METHOD ErrorHandler : BOOL
VAR_INPUT
END_VAR
VAR
END_VAR
//once error scanned
IF currentMode = eOperationModes.AUTO THEN
	//once error deteted and in AUTO mode , forcely switch to SEMI_AUTO
	currentMode := eOperationModes.SEMI_AUTO;
END_IF
//reset error handling
IF requestErrorClear <> eErrorClearWays.NO_ACTION THEN
	errorDevice^.ErrorClear(requestErrorClear); //call error clear function
	requestErrorClear := eErrorClearWays.NO_ACTION;
	errorDevice := 0 ;// cut link
END_IF
END_METHOD

METHOD FB_init : BOOL
VAR_INPUT
	bInitRetains : BOOL; // if TRUE, the retain variables are initialized (warm start / cold start)
	bInCopyCode : BOOL;  // if TRUE, the instance afterwards gets moved into the copy code (online change)
	
	argParent : POINTER TO RunUnitGeneric;
	argSlotBase : POINTER TO RunMaterial;
	argSlotLast : POINTER TO RunMaterial;
	
	argPbRed : POINTER TO RunSignal;
	argPbGreen : POINTER TO RunSignal;
	argPbYellow : POINTER TO RunSignal;
	
	argInterfaceControl : POINTER TO InterfaceControlV1;
	argInterfaceManual : POINTER TO InterfaceManualV1;
END_VAR
//initialize 
Parent := argParent;
SlotBase := argSlotBase;
SlotLast := argSlotLast;
//
IF bInitRetains THEN
	NextState := eSpecialStates.INITIAL_BEGIN;
END_IF
//input
pbRed := argPbRed;
pbGreen := argPbGreen;
pbYellow := argPbYellow;

interfaceControl := argInterfaceControl;
interfaceManual := argInterfaceManual;

interfaceControl^.state := TO_WORD(eSpecialStates.MAIN_WAIT_INITIALIZING);
END_METHOD

METHOD Initialize : BOOL
VAR_INPUT
END_VAR
END_METHOD

END_FUNCTION_BLOCK

// ---- POUs/Foundation/RunUnitIndexerMaster.TcPOU
FUNCTION_BLOCK RunUnitIndexerMaster EXTENDS RunUnitTransporterBase
VAR		
	Axis : POINTER TO RunAxis; //axis reference
	
	//Working registers
	nCounter : DINT;
	
	
END_VAR
VAR PERSISTENT
END_VAR

SUPER^(); // call base class's execution

//---------------
//	S16#0-S16#0F : regular state as standard indexer
//	S16#10 : mechanical control of movement
//---------------

IF NOT workingTimer.IN THEN
	 workingTimer.IN := TRUE;
END_IF

CASE outputState OF
	16#0:
		//-------------------------
		//	Trigger all slaves
		//-------------------------
		FOR nCounter:=1 TO 4 BY 1 DO
			slaveWorkingSignal[nCounter] := slaveLinkageStatus[nCounter];
		END_FOR
		bSerialTransition := TRUE;
		
		THIS^.workingTimerCache := THIS^.workingTimer.ET;
		workingTimer.IN := FALSE; //reset
	16#1:	
		//------------------------------------------
		//check material synchronization to Databse
		//All slot act must be off
		//------------------------------------------
		bSerialTransition := TRUE;
		FOR nCounter:=0 TO SlotCount-1 BY 1 DO
			bSerialTransition := bSerialTransition AND NOT SlotBase[nCounter].Act;
		END_FOR
	16#2:
		//--------------------------------
		// Scanning working signal until all are off
		//--------------------------------
		bSerialTransition := TRUE;
		FOR nCounter:= 1 TO 32 BY 1 DO
			bSerialTransition := bSerialTransition AND NOT slaveWorkingSignal[nCounter];
		END_FOR
	16#3:
		//-------------------
		//Sync with down stream
		//-------------------
		IF syncEngaged AND syncAcknowledged THEN
			syncEngaged := FALSE; //reset
		END_IF
		bSerialTransition := NOT syncAcknowledged; //make sure signal is resetted
		IF bSerialTransition THEN
			//move last slot's information to buffer area
			syncMatId:= SlotLast^.Id; // for the last slot
			syncMatValid := SlotLast^.Valid;// ready to sync
		END_IF
	16#4:
		//2 modes
		// a. synchronize with downstream only, go with pull upstream if avialable
		// b. synchronize with down/upstream both
	
		// pull by downstream (set on then check off
		// pull upstream (check on then reset
		
		IF syncMatValid AND NOT syncEngaged THEN
			syncEngaged := TRUE;//ready to synchronizing (communicate with downstream
		END_IF
		
		//listen to move
		bSerialTransition :=  (NOT syncMatValid) OR (syncAcknowledged AND syncMatValid);
		IF bSerialTransition THEN
			NextState := 16#10;
		END_IF
	16#10:
		//---------------------
		//shifting movement mechaincal
		//---------------------	
	16#F:
		//---------------------------------------------------------------
		//Do data shifting (move is valid/id) , leave first slot as empty
		//---------------------------------------------------------------
		FOR nCounter:=SlotCount-1 TO 0 BY -1 DO
			IF nCounter > 0 THEN
				SlotBase[nCounter].Id := SlotBase[nCounter-1].id;
				SlotBase[nCounter].Valid := SlotBase[nCounter-1].Valid;
			END_IF			
		END_FOR
		NextState := 16#0;
END_CASE

METHOD FB_init : BOOL
VAR_INPUT
	bInitRetains : BOOL; // if TRUE, the retain variables are initialized (warm start / cold start)
	bInCopyCode : BOOL;  // if TRUE, the instance afterwards gets moved into the copy code (online change)
	
	argParent : POINTER TO RunUnitGeneric;
	argSlotBase : POINTER TO RunMaterial;
	argSlotLast : POINTER TO RunMaterial;
	
	argUpstream : POINTER TO RunUnitTransporterBase;
	argAxis : POINTER TO RunAxis;

END_VAR
//initialize 
Parent := argParent;
SlotBase := argSlotBase;
SlotLast := argSlotLast;

Axis := argAxis;
Upstream := argUpstream;

IF Upstream=0 THEN
	isProxyMode:=TRUE; //no upstream , i am proxy
END_IF

//calculate how much slot related
SlotCount :=  TO_INT((SlotLast-SlotBase)/SIZEOF(RunMaterial) + 1);
END_METHOD

END_FUNCTION_BLOCK

// ---- POUs/Foundation/RunUnitTransporterBase.TcPOU
FUNCTION_BLOCK RunUnitTransporterBase EXTENDS RunUnitGeneric
VAR_INPUT	
	//self
	syncAcknowledged AT%M*  : BOOL; //downstream replied starting ackowledge , face to downstream
	syncMatId AT%M* : DWORD := 0;
	syncMatValid AT%M* : BOOL := FALSE;
END_VAR
VAR_OUTPUT
	//self
	syncEngaged AT%M*  : BOOL; //inform downstream i am ready , face to downstream
	
END_VAR
VAR		
	//
	Upstream : POINTER TO RunUnitTransporterBase;//upstream linkage
	//proxy mode
	isProxyMode : BOOL := FALSE;
	
	pollingTimer : TON;
	fbAdsSyncRead : FB_ReadAdsSymByName;
	fbAdsSyncWrite : FB_WriteAdsSymByName;
	fbAdsSyncMatIdRead : FB_ReadAdsSymByName;
	fbAdsSyncMatValidRead : FB_ReadAdsSymByName;
	
	preSyncEngaged : BOOL := FALSE;
	
END_VAR
VAR PERSISTENT
	//proxy mode parameters
	netId : T_AmsNetID;
	port : T_AmsPort := 851; //Tc3
	
	varNameSyncEngaged : STRING;
	varNameSyncAckowledged : STRING;
	varNameSyncMatIdSync : STRING;
	varNameSyncMatValidSync : STRING;
END_VAR

//non proxy 	
SUPER^();

IF (outputState <> NextState) OR bSerialTransition THEN
	//once state transit , reset timer
	timeoutTimer.IN := FALSE;
ELSIF NOT timeoutTimer.IN THEN
	//once timer not activated 
	timeoutTimer.IN := TRUE;
END_IF

IF NOT isProxyMode THEN
	RETURN;
END_IF

pollingTimer(IN:= NOT pollingTimer.Q, PT:= T#50MS, Q=> , ET=> );

//do ADS data exchanging
fbAdsSyncRead(
	bRead:= pollingTimer.Q and not fbAdsSyncRead.bBusy, 
	sNetId:= netId, 
	nPort:= port, 
	sVarName:= varNameSyncEngaged, 
	nDestAddr:= ADR(preSyncEngaged), 
	nLen:= SIZEOF(preSyncEngaged), 
	tTimeout:= , 
	eComMode:= , 
	bBusy=> , 
	bError=> , 
	nErrorId=> );
		
fbAdsSyncWrite(
	bWrite:= pollingTimer.Q AND NOT fbAdsSyncWrite.bBusy, 
	sNetId:= netId, 
	nPort:= port, 
	sVarName:= varNameSyncAckowledged, 
	nSrcAddr:= ADR(syncAcknowledged), 
	nLen:= SIZEOF(syncAcknowledged), 
	tTimeout:= , 
	eComMode:= , 
	bBusy=> , 
	bError=> , 
	nErrorId=> );		
			
fbAdsSyncMatIdRead(
	bRead:= , 
	sNetId:= netId, 
	nPort:= port, 
	sVarName:= varNameSyncMatIdSync, 
	nDestAddr:= ADR(syncMatId), 
	nLen:= SIZEOF(syncMatId), 
	tTimeout:= , 
	eComMode:= , 
	bBusy=> , 
	bError=> , 
	nErrorId=> );
fbAdsSyncMatValidRead(
	bRead:= , 
	sNetId:= netId, 
	nPort:= port, 
	sVarName:= varNameSyncMatValidSync, 
	nDestAddr:= ADR(syncMatValid), 
	nLen:= SIZEOF(syncMatValid), 
	tTimeout:= , 
	eComMode:= , 
	bBusy=> , 
	bError=> , 
	nErrorId=> );
	

//data exchanging do not be break
atomicOperation := TRUE;
CASE outputState OF
	0:
		IF preSyncEngaged THEN
						
			//start reading
			fbAdsSyncMatIdRead.bRead := TRUE;
			fbAdsSyncMatValidRead.bRead:= TRUE;
			
			bSerialTransition := TRUE;
		END_IF
	1:
		IF NOT fbAdsSyncMatIdRead.bBusy AND NOT fbAdsSyncMatValidRead.bBusy THEN
			syncEngaged:= TRUE; //mat sync verified , output to downstream
			bSerialTransition := TRUE;
		END_IF
	2: 
		IF NOT preSyncEngaged THEN
			//done
			syncEngaged := FALSE;
			//wait for next reading
			fbAdsSyncMatIdRead.bRead := FALSE;
			fbAdsSyncMatValidRead.bRead:= FALSE;
			
			
			NextState := 0;
		END_IF
END_CASE

METHOD FB_init : BOOL
VAR_INPUT
	bInitRetains : BOOL; // if TRUE, the retain variables are initialized (warm start / cold start)
	bInCopyCode : BOOL;  // if TRUE, the instance afterwards gets moved into the copy code (online change)
	
	argParent : POINTER TO RunUnitGeneric;
	argSlotBase : POINTER TO RunMaterial;
	argSlotLast : POINTER TO RunMaterial;
	
	argUpstream : POINTER TO RunUnitTransporterBase;
END_VAR
//initialize 
Parent := argParent;
SlotBase := argSlotBase;
SlotLast := argSlotLast;

Upstream := argUpstream;

IF Upstream=0 THEN
	isProxyMode:=TRUE; //no upstream , i am proxy
END_IF
END_METHOD

METHOD Initialize : BOOL
VAR_INPUT
END_VAR

//reset sync signal
CASE outputState OF
	eSpecialStates.INITIAL_BEGIN:
		syncEngaged := FALSE; //reset
		IF Upstream <> 0 THEN
			Upstream^.syncAcknowledged := FALSE; //reset
		END_IF
		//direct change state
		NextState := eSpecialStates.INITIAL_END;
END_CASE

Initialize := SUPER^.Initialize();
END_METHOD

END_FUNCTION_BLOCK

// ---- POUs/IncNoOverflow.TcPOU
FUNCTION IncNoOverflow : UDINT
VAR_INPUT
	input : UDINT;
END_VAR
VAR
END_VAR

IF input >= 16#FFFFFFFF THEN
	IncNoOverflow := 0;
ELSE
	IncNoOverflow := input +1;
END_IF

END_FUNCTION

// ---- POUs/MAIN.TcPOU
PROGRAM MAIN
VAR

cbBlock1 : CommandBlockBase;
cbBlock2 : CommandBlockBase;

cbBlock3 : CommandBlockPos;
cbBlock4 : CommandBlockPos;

ptBlock : POINTER TO CommandBlockBase := ADR(cbBlock1);	
ptBlockPos : POINTER TO CommandBlockPos;

aSize : INT;


memoryPool : ARRAY[1..1024] OF WORD;

ptRunIndexerMaster : POINTER TO RunUnitIndexerMaster;
ptRunGeneric : POINTER TO RunUnitGeneric;

ptUnitGeneric : POINTER TO UnitBase;
ptUnitIndexerMaster : POINTER TO UnitIndexerMaster;

bInitialized : BOOL ;
nCounter : int ;
END_VAR

cbBlock1.AXIS_ID:=5;
MAIN.ptBlock:=ADR(cbBlock1);

cbBlock2:=MAIN.ptBlock^; // value assignment?
//change cbBlock1 , watch if cbBlock2 changed

MAIN.ptBlock := ADR(cbBlock3); //if possible mophism

cbBlock3.COORDINATE:=1234;

ptBlockPos:=MAIN.ptBlock;
cbBlock4:=ptBlockPos^;//check


//may access violation??
//ptBlockPos:=ADR(cbBlock1);
//ptBlockPos^.COORDINATE:=5555; //may violation

//TEST2();
//TEST_CYLINDER();
//TEST_UNIT_VIRTUAL();
//TEST_UNIT_MASTER();
//TEST_AXIS();
IF NOT bInitialized THEN
	FOR nCounter:=8 TO 10 BY 1 DO
		GVL.commandBlocks[nCounter].command := eCommandTypes.POSITION;
		GVL.commandBlocks[nCounter].parameter.position.Acceleration := 4000;
		GVL.commandBlocks[nCounter].parameter.position.Deceleration := 4000;

	END_FOR
	GVL.commandBlocks[8].parameter.position.Position := 300;
	GVL.commandBlocks[8].parameter.position.Velocity := 400;
	
	GVL.commandBlocks[9].parameter.position.Position := 400;
	GVL.commandBlocks[9].parameter.position.Velocity := 100;
	
	GVL.commandBlocks[10].parameter.position.Position := 800;
	GVL.commandBlocks[10].parameter.position.Velocity := 400;
	
	bInitialized := true;
END_IF
TEST_BUFFERING();

aSize := SIZEOF(GVL.unitControls[1]);
aSize := SIZEOF(UnitBase);
aSize := SIZEOF(UnitIndexerMaster);
//fbCylinder(ptBlock:= ADR(cylinderBlock));

//fbRunIndexerMaster(ptBlock:= );


//no need
//ptRunIndexerMaster := ADR(memoryPool[1]); // fine?
//ptRunGeneric := ADR(memoryPool[1+SIZEOF(ptRunIndexerMaster)]);

//ptRunIndexerMaster^();
//ptRunGeneric^();


//possible manipulate memory allocation
ptUnitGeneric := ADR(memoryPool[1]);
ptUnitIndexerMaster := ADR(memoryPool[1+SIZEOF(ptUnitGeneric^)]);

ptUnitGeneric^.alarmCode := 99;  //

METHOD FB_init : BOOL
VAR_INPUT
	bInitRetains : BOOL; // if TRUE, the retain variables are initialized (warm start / cold start)
	bInCopyCode : BOOL;  // if TRUE, the instance afterwards gets moved into the copy code (online change)
END_VAR
END_METHOD

END_PROGRAM

// ---- POUs/Stations/CellularD/RunCableHolder.TcPOU
FUNCTION_BLOCK RunCableHolder EXTENDS RunUnitSlave
VAR
	//devices
	holderFixedEnd : POINTER TO RunCylinder;
	holderMovingEnd : POINTER TO RunCylinder;
	shifterShort : POINTER TO RunCylinder;
	shifterLong : POINTER TO RunCylinder;
	//axis (share
	axis : POINTER TO RunAxis;
	ptDrag : POINTER TO ParameterSet;
	ptRelease : pointer to ParameterSet;
END_VAR

SUPER^();

CASE outputState OF
	//---------------Initialize
	eSpecialStates.INITIAL_BEGIN:
		transitionByte.0 :=  holderFixedEnd^.Execute(eCylinderCommands.COMMAND_A);
		transitionByte.1 :=  holderMovingEnd^.Execute(eCylinderCommands.COMMAND_A);
		transitionByte.2 :=  shifterShort^.Execute(eCylinderCommands.COMMAND_A);
		transitionByte.3 :=  shifterLong^.Execute(eCylinderCommands.COMMAND_A);
		IF transitionByte = 16#F THEN
			NextState := eSpecialStates.INITIAL_END;
		END_IF
	//---------------Working
	eSpecialStates.SLAVE_ENTER_PROCEDURE:
		IF bMaterialOverride THEN
			bSerialTransition := TRUE;
		ELSE
			NextState := eSpecialStates.SLAVE_WORK_DONE;	
		END_IF
		//TODO , check ok/ng?
	16#201:
		bSerialTransition := shifterLong^.Execute(eCylinderCommands.COMMAND_B);
	16#202:
		//hold
		transitionByte.0 :=  holderFixedEnd^.Execute(eCylinderCommands.COMMAND_B);
		transitionByte.1 :=  holderMovingEnd^.Execute(eCylinderCommands.COMMAND_B);
		bSerialTransition := (transitionByte = 16#3);
	16#203:
		bSerialTransition := axis^.ExecuteParameter(ptDrag);//inform transporter moving work2
	16#204:
		//strech
		IF shifterShort^.Execute(eCylinderCommands.COMMAND_B) THEN
			slaveWorkingSignal[1] := TRUE; //inform to labeler handler to work
			NextState := 16#210;
		END_IF
	//-------------Releasing
	16#210:
		//wait until
		bSerialTransition := NOT slaveWorkingSignal[1];
	16#211:
		transitionByte.0 := holderFixedEnd^.Execute(eCylinderCommands.COMMAND_A); //release
		transitionByte.1 := holderMovingEnd^.Execute(eCylinderCommands.COMMAND_A);
		IF transitionByte = 16#3 THEN
			bSerialTransition := TRUE;
		END_IF
	16#212:
		bSerialTransition := axis^.ExecuteParameter(ptRelease);//inform transporter moving release
	16#213:
		//release
		bSerialTransition := shifterLong^.Execute(eCylinderCommands.COMMAND_A);
	16#214:
		//release
		bSerialTransition := holderMovingEnd^.Execute(eCylinderCommands.COMMAND_A);
	16#215:
		IF shifterShort^.Execute(eCylinderCommands.COMMAND_A) THEN
			NextState := eSpecialStates.SLAVE_WORK_DONE; //rewind
		END_IF
END_CASE

METHOD FB_init : BOOL
VAR_INPUT
	bInitRetains : BOOL; // if TRUE, the retain variables are initialized (warm start / cold start)
	bInCopyCode : BOOL;  // if TRUE, the instance afterwards gets moved into the copy code (online change)
	
	argParent : POINTER TO RunUnitGeneric;
	argSlotBase : POINTER TO RunMaterial;
	argSlotLast : POINTER TO RunMaterial;
	
	argWorkingSignal : POINTER TO BOOL;
	
	//devices
	argHolderFixedEnd : POINTER TO RunCylinder;
	argHolderMovingEnd : POINTER TO RunCylinder;
	argShifterShort : POINTER TO RunCylinder;
	argShifterLong : POINTER TO RunCylinder;
	
	//
	argAxis : POINTER TO RunAxis;
END_VAR
VAR CONSTANT
	indexDrag : INT :=8;
	indexRelease : int :=9;
END_VAR
//initialize 
Parent := argParent;
SlotBase := argSlotBase;
SlotLast := argSlotLast;
//
IF bInitRetains THEN
	NextState := eSpecialStates.INITIAL_BEGIN;
END_IF

workingSignal := argWorkingSignal; //link

//device link
holderFixedEnd := argHolderFixedEnd;
holderMovingEnd := argHolderMovingEnd;
shifterShort := argShifterShort;
shifterLong := argShifterLong;

//
axis := argAxis;
ptDrag := ADR(axis^.ptpCommands[indexDrag]);
ptRelease := ADR(axis^.ptpCommands[indexRelease]);
END_METHOD

END_FUNCTION_BLOCK

// ---- POUs/Stations/CellularD/RunGradeOutput.TcPOU
FUNCTION_BLOCK RunGradeOutput EXTENDS RunUnitSlave
VAR
	axisMoving : POINTER TO RunAxis;
	holder : POINTER TO RunCylinder;
	axisVertical : POINTER TO RunCylinder;
	clamper : POINTER TO RunCylinder;	
	//
	ptCommandReady : POINTER TO ParameterSet;
	ptCommandOK : POINTER TO ParameterSet;
	ptCommandNG : POINTER TO ParameterSet;
	//
	block : MaterialBlock;
	ptDesitination : POINTER TO parameterset;
END_VAR
VAR PERSISTENT
	isQuery : bool ; //whether query material data when material income
END_VAR

//Ng/OK output mechanism
SUPER^();

CASE outputState OF 
	//-------------------------Initialize
	eSpecialStates.INITIAL_BEGIN:
		transitionByte.0 := holder^.Execute(eCylinderCommands.COMMAND_A);
		transitionByte.1 := clamper^.Execute(eCylinderCommands.COMMAND_A);
		bSerialTransition := (transitionByte = 16#3);
	eSpecialStates.INITIAL_STATE_1:
		bSerialTransition :=  axisVertical^.Execute(eCylinderCommands.COMMAND_A);
	eSpecialStates.INITIAL_STATE_2:
		IF axisMoving^.ExecuteParameter(ptCommandReady) THEN
			NextState := eSpecialStates.INITIAL_END;
		END_IF
	//------------------------Working
	eSpecialStates.SLAVE_ENTER_PROCEDURE:
		//---------------
		//	Material infor exchanging
		//---------------
		SlotLast^.Id := SlotBase^.Id; //the clamper work station
		SlotLast^.Valid := SlotLast^.Valid;
		IF SlotLast^.Valid THEN
			SlotLast^.Act := isQuery; //query grade
			bSerialTransition := TRUE;
		ELSE
			NextState := eSpecialStates.SLAVE_WORK_DONE;		
		END_IF
	16#201:
		bSerialTransition:=axisVertical^.Execute(eCylinderCommands.COMMAND_B); //down
	16#202:
		bSerialTransition:=holder^.Execute(eCylinderCommands.COMMAND_B); //hold
	16#203:
		bSerialTransition:=clamper^.Execute(eCylinderCommands.COMMAND_B); //clamper relase
	16#204:
		bSerialTransition:=axisVertical^.Execute(eCylinderCommands.COMMAND_A); //up
	16#205:
		bSerialTransition:=clamper^.Execute(eCylinderCommands.COMMAND_A); //clamper return
		IF bSerialTransition THEN
			workingSignal^ := FALSE; //release conveyor
		END_IF
	16#206:
		bSerialTransition := NOT SlotLast^.Act; //wait until query over
		IF bSerialTransition THEN
			block := SlotLast^.Data;
			CASE block.data[0] OF
				0:
					//ng
					ptDesitination := ptCommandNG;
				1:
					//ok
					ptDesitination := ptCommandOK;
			END_CASE
		END_IF
	16#207:
		IF axisMoving^.ExecuteParameter(ptDesitination) THEN
			//according TO grade TO MOVE
			NextState := 16#210;
		END_IF
	//-------------------Drop
	16#210: 
		bSerialTransition:=holder^.Execute(eCylinderCommands.COMMAND_A); //release
	16#211:
		IF axisMoving^.ExecuteParameter(ptCommandReady) THEN
			NextState := 0;
		END_IF
END_CASE

METHOD FB_init : BOOL
VAR_INPUT
	bInitRetains : BOOL; // if TRUE, the retain variables are initialized (warm start / cold start)
	bInCopyCode : BOOL;  // if TRUE, the instance afterwards gets moved into the copy code (online change)
	
	argParent : POINTER TO RunUnitGeneric;
	argSlotBase : POINTER TO RunMaterial;
	argSlotLast : POINTER TO RunMaterial;
	
	argWorkingSignal : POINTER TO BOOL;
	
	argAxisMoving : POINTER TO RunAxis;
	
	argHolder : POINTER TO RunCylinder;
	argAxisVertical : POINTER TO RunCylinder;
	argClamper : POINTER TO RunCylinder;
	
END_VAR
VAR CONSTANT
	indexReady : INT := 1;
	indexOK : INT := 2;
	indexNG : INT := 3;
END_VAR
//initialize 
Parent := argParent;
SlotBase := argSlotBase;
SlotLast := argSlotLast;
//
IF bInitRetains THEN
	NextState := eSpecialStates.INITIAL_BEGIN;
END_IF

workingSignal := argWorkingSignal; //link

//Axis
axisMoving := argAxisMoving;
ptCommandReady := ADR(axisMoving^.ptpCommands[indexReady]);
ptCommandOK := ADR(axisMoving^.ptpCommands[indexOK]);
ptCommandNG := ADR(axisMoving^.ptpCommands[indexNG]);

holder := argHolder;
axisVertical := argAxisVertical;
clamper := argClamper;
END_METHOD

END_FUNCTION_BLOCK

// ---- POUs/Stations/CellularD/RunLabelHandler.TcPOU
FUNCTION_BLOCK RunLabelHandler EXTENDS RunUnitSlave
VAR_INPUT
END_VAR
VAR_OUTPUT
END_VAR
VAR
	//File handler
	fbOpen : FB_FileOpen;
	fbWrite : FB_FileWrite;
	fbClose : FB_FileClose;
	fileHandle : UINT;
	
	fileContent : STRING := '100,2';
	fileBytes : ARRAY[0..15] OF BYTE;
	// communicate with external device
	ioPrinter : POINTER TO  ioBundlePrinterApplicator;
	// Vaccuum
	ioVacuum : POINTER TO ioBundleLabelGripper;
	bVacuumSensor : POINTER TO RunSignal;
	//
	axis : POINTER TO RunAxis;
	//
	gripperVertical : POINTER TO RunCylinder;
	gripperRotate : POINTER TO RunCylinder;
	gripperPressorVertical : POINTER TO RunCylinder;
	gripperPressorPress : POINTER TO RunCylinder;
	shifter : POINTER TO RunCylinder;
	//
	ptCommandReady : POINTER TO ParameterSet;
	ptCommandLabelTake : POINTER TO ParameterSet;
	ptCommandLabelPlace : POINTER TO ParameterSet;
	//
	pressCounter : INT := 0;
	//
	bFirstCycle : bool := false;
END_VAR
VAR PERSISTENT
	bVacuumTimeout : TON;
	pressGoal : INT := 3;
	filePath : STRING := '';
	printerStartDurance : TON;
END_VAR

SUPER^();

//auto reset printer-start signal
printerStartDurance(IN:= ioPrinter^.prtStart, PT:= , Q=> , ET=> );
IF ioPrinter^.prtStart AND printerStartDurance.Q THEN
	ioPrinter^.prtStart := FALSE; // auto off
END_IF

//into initial state
IF NOT bFirstCycle AND outputState=0 THEN
	NextState := 16#300;
	bFirstCycle := TRUE;
END_IF

CASE outputState OF 
	//-------------------Initializing
	eSpecialStates.INITIAL_BEGIN:
		//all cylinder off
		transitionByte.0 := gripperVertical^.Execute(eCylinderCommands.COMMAND_A);
		transitionByte.1 := gripperRotate^.Execute(eCylinderCommands.COMMAND_A);
		transitionByte.2 := gripperPressorVertical^.Execute(eCylinderCommands.COMMAND_A);
		transitionByte.3 := gripperPressorPress^.Execute(eCylinderCommands.COMMAND_A);
		transitionByte.4 := shifter^.Execute(eCylinderCommands.COMMAND_A);
		bSerialTransition := (transitionByte = 16#1F);
	eSpecialStates.INITIAL_STATE_1:
		bSerialTransition := axis^.ExecuteParameter(ptCommandReady);
	eSpecialStates.INITIAL_STATE_2:
		IF ioPrinter^.prtData THEN
			ioPrinter^.prtStart := TRUE; //clear all cached data
		ELSE
			//no data remained , go ahead
			bFirstCycle := FALSE;
			NextState := eSpecialStates.INITIAL_END;
		END_IF
	//-------------------Working
	16#300:
		//TODO , label printing triggered by HMI , according to the data from DB
		fbOpen.bExecute:=TRUE;
		bSerialTransition := TRUE;
	16#301:
		bSerialTransition := NOT fbOpen.bBusy;
		IF bSerialTransition THEN
			fbOpen.bExecute:=FALSE;
		END_IF
	16#302:
		fbWrite.bExecute := TRUE;
		bSerialTransition := TRUE;
	16#303:
		bSerialTransition := NOT fbWrite.bBusy;
		IF bSerialTransition THEN
			fbWrite.bExecute:=FALSE;
		END_IF
	16#304:
		fbClose.bExecute := TRUE;
		bSerialTransition := TRUE;
	16#305:
		IF NOT fbClose.bBusy THEN
			fbClose.bExecute := false;
			NextState:=16#400;
		END_IF
	//-----------------------------
	16#400:
		bSerialTransition := ioPrinter^.prtData;
		IF bSerialTransition THEN
			ioPrinter^.prtStart := TRUE;
		END_IF
	16#401:
		//waiting printer
		bSerialTransition := NOT ioPrinter^.prtEnd AND NOT ioPrinter^.prtData ;
	16#402:
		bSerialTransition := axis^.ExecuteParameter(ptCommandLabelTake);
	16#403:
		bSerialTransition := gripperVertical^.Execute(eCylinderCommands.COMMAND_B);	//down
		IF bSerialTransition THEN
			//generate vacuum
			ioVacuum^.vacuumGripper := TRUE; //on
			ioVacuum^.breakGripper := FALSE;
			//
			bVacuumTimeout.IN :=TRUE;
		END_IF
	16#404:
		bSerialTransition := bVacuumSensor^.debouncedOn;
		IF bSerialTransition THEN
			bVacuumTimeout.IN :=FALSE; //reset
		ELSIF bVacuumTimeout.Q THEN
			//TODO , timeout alarm
		END_IF
	16#405:
		bSerialTransition := gripperVertical^.Execute(eCylinderCommands.COMMAND_A); //up
	16#406:
		IF axis^.ExecuteParameter(ptCommandLabelPlace) THEN
			//up
			NextState := 0; //wait trigger
		END_IF
	//-----------------Tag
	eSpecialStates.SLAVE_ENTER_PROCEDURE:
		bSerialTransition := gripperVertical^.Execute(eCylinderCommands.COMMAND_B); //down
		IF bSerialTransition THEN
			//break vacuum
			ioVacuum^.vacuumGripper := FALSE; //off
			ioVacuum^.breakGripper := TRUE;
		END_IF
	16#201:
		transitionByte.0 := gripperVertical^.Execute(eCylinderCommands.COMMAND_A); //up
		transitionByte.1 := gripperRotate^.Execute(eCylinderCommands.COMMAND_A); //back
		bSerialTransition := (transitionByte = 16#3);
	//----------------Press
	16#202:
		bSerialTransition := shifter^.Execute(eCylinderCommands.COMMAND_B); //tool change
	16#203:
		bSerialTransition := gripperPressorVertical^.Execute(eCylinderCommands.COMMAND_B); //down
	16#204:
		bSerialTransition := gripperPressorPress^.Execute(eCylinderCommands.COMMAND_B);
	16#205:
		IF gripperPressorPress^.Execute(eCylinderCommands.COMMAND_A) THEN
			pressCounter := pressCounter+1;
			
			IF pressCounter >= pressGoal THEN
				//press back-forth
				NextState := 16#230;
			ELSE
				NextState := 16#205;
			END_IF
		END_IF
	//------------Return
	16#230:
		bSerialTransition := gripperPressorVertical^.Execute(eCylinderCommands.COMMAND_A); //up
	16#231:
		bSerialTransition := shifter^.Execute(eCylinderCommands.COMMAND_A); //up
		IF bSerialTransition THEN
			workingSignal^ := FALSE; //off
			bWorkingOverride:= false;
		END_IF
	16#232:
		//ready
		IF axis^.ExecuteParameter(ptCommandLabelTake) THEN
			pressCounter:=0;
			NextState := 16#300;
		END_IF
END_CASE
bVacuumTimeout(IN:= , PT:= , Q=> , ET=> );


//file 
fbOpen(
	sNetId:= , 
	sPathName:= filePath, 
	nMode:= FOPEN_MODEWRITE, 
	ePath:= , 
	bExecute:= , 
	tTimeout:= , 
	bBusy=> , 
	bError=> , 
	nErrId=> , 
	hFile=> fileHandle);
fbWrite(
	sNetId:= , 
	hFile:= fileHandle, 
	pWriteBuff:= ADR(fileBytes), 
	cbWriteLen:= SIZEOF(fileBytes), 
	bExecute:= , 
	tTimeout:= , 
	bBusy=> , 
	bError=> , 
	nErrId=> , 
	cbWrite=> );
fbClose(
	sNetId:= , 
	hFile:= fileHandle, 
	bExecute:= , 
	tTimeout:= , 
	bBusy=> , 
	bError=> , 
	nErrId=> );

METHOD FB_init : BOOL
VAR_INPUT
	bInitRetains : BOOL; // if TRUE, the retain variables are initialized (warm start / cold start)
	bInCopyCode : BOOL;  // if TRUE, the instance afterwards gets moved into the copy code (online change)
	
	argParent : POINTER TO RunUnitGeneric;
	argSlotBase : POINTER TO RunMaterial;
	argSlotLast : POINTER TO RunMaterial;
	
	argWorkingSignal : POINTER TO BOOL;
	
	//devices
	argVacuumSensor : POINTER TO RunSignal;
	
	argAxis : POINTER TO RunAxis;
	//
	argGripperVertical : POINTER TO RunCylinder;
	argGripperRotate : POINTER TO RunCylinder;
	argGripperPressorVertical : POINTER TO RunCylinder;
	argGripperPressorPress : POINTER TO RunCylinder;
	argShifter : POINTER TO RunCylinder;
	//
	argIoPrinter : POINTER TO ioBundlePrinterApplicator;
	argIoVacuum : POINTER TO ioBundleLabelGripper;
END_VAR
VAR CONSTANT
	indexReady : INT := 1;
	indexTake :INT :=2;
	indexPlace : INT :=3;
END_VAR
//initialize 
Parent := argParent;
SlotBase := argSlotBase;
SlotLast := argSlotLast;
//
IF bInitRetains THEN
	NextState := eSpecialStates.INITIAL_BEGIN;
END_IF

workingSignal := argWorkingSignal; //link

//device link
//
axis := argAxis;
//
gripperVertical := argGripperVertical;
gripperRotate := argGripperRotate;
gripperPressorVertical := argGripperPressorVertical;
gripperPressorPress := argGripperPressorPress;
shifter := argShifter;

ptCommandReady := ADR(axis^.ptpCommands[indexReady]);
ptCommandLabelTake := ADR(axis^.ptpCommands[indexTake]);
ptCommandLabelPlace := ADR(axis^.ptpCommands[indexPlace]);

bVacuumSensor := argVacuumSensor;

ioPrinter := argIoPrinter;
ioVacuum := argIoVacuum;
END_METHOD

END_FUNCTION_BLOCK

// ---- POUs/Stations/HRASI/InitAndTaskControl/RunCoordinator.TcPOU
FUNCTION_BLOCK RunCoordinator EXTENDS RunGroupNode
VAR_INPUT
	commStartProductionMode AT%M* : BOOL;
	commStartRegularCheckMode AT%M* : BOOL;
	commIsDryRun AT%M* : BOOL;
	//------------
	//	Trial mode
	//------------
	commStartTrialAssemble AT%M* : BOOL;
	commStartTrialSnap AT%M* : BOOL;
	//------------
	// link to HMI
	//------------
	commRegularCheckAck AT%I* : BOOL;
	//------------
	//	Control
	//------------
	scara1 : POINTER TO RunScaraAgent;
	scara2 : POINTER TO RunScaraAgent;
	
	clamper1 : POINTER TO RunClamper;
	clamper2 : POINTER TO RunClamper;
	
	loader : POINTER TO RunLoading;
	aoi : POINTER TO RunAoiInspectionV1;
	
	bridge1 : POINTER TO RunBridge;
	
	racks : ARRAY[0..3] OF POINTER TO RunCommonRack;
END_VAR
VAR_OUTPUT
	isInitialized AT%Q*: BOOL;
	isIdle AT%Q* : BOOL;
END_VAR
VAR
	dryRunDevicesList : ARRAY[0..7] OF POINTER TO executebase;
	
	//Vacuum breaker
	backSecureBreaker AT%Q* : BOOL;
	filterBreaker AT%Q* : BOOL;
	
END_VAR
VAR PERSISTENT 
	commSpeedFactor AT%M* : BYTE;
	timerBreak : ton;
END_VAR
VAR CONSTANT 
	ERR_VACUUM_JAMMED : DWORD := 600;
END_VAR

//Initialization sequences:
// 1. Group1 - two clamper and indexer (two clamper hold/unhold , the indexer turing 4 runs)
// 2. Group2 - SCARA1 and rack1,2 (pick to drop zone then homing and release rackes)
// 3. Group3 - SCARA2 and rack3,4

SUPER^();
timerBreak();

isInitialized := ((outputState AND eSpecialStates.INITIAL_REGION) <> 16#100);
isIdle := outputState = eSpecialStates.GENERIC_GROUP_IDLE;

IF dryRunDevicesList[0] = 0 THEN
	//initialize
	dryRunDevicesList[0] := ADR(gvl.vacuumControls[A9]); 
	dryRunDevicesList[1] := ADR(gvl.vacuumControls[A10]);
	dryRunDevicesList[2] := ADR(gvl.vacuumControls[A11]);
	dryRunDevicesList[3] := ADR(gvl.vacuumControls[A12]);
	
	dryRunDevicesList[4] := ADR(gvl.vacuumControls[A13]);
	dryRunDevicesList[5] := ADR(gvl.vacuumControls[A14]);

	dryRunDevicesList[6] := ADR(gvl.vacuumControls[A20]);
	
	dryRunDevicesList[7] := ADR(gvl.cylinderControls[cy6]); //top part clamper
	
END_IF

CASE outputState OF
	//----------------------------
	//	Initializing :
	// 1. Off all I/O 
	// 2. SCARA & Clamper & Indexer
	//----------------------------
	eSpecialStates.INITIAL_BEGIN:
		commStartProductionMode := FALSE;
		commStartRegularCheckMode :=FALSE;
		commIsDryRun := FALSE;
		commStartTrialAssemble:=FALSE;
		commStartTrialSnap:=FALSE;
		commRegularCheckAck:=FALSE;
		isPurged := FALSE;
		
		THIS^.TurnDryRun(FALSE);
		loader^.isWorking := FALSE;
		
		bSerialTransition := TRUE;
	//-----------------------------
	// Off remote I/O devices
	//-----------------------------
	eSpecialStates.INITIAL_STATE_1:
		bSerialTransition:=TRUE;
		FOR nCounter :=0 TO 23 BY 1 DO
			IF gvl.remoteControls[nCounter] <> 0 THEN
				bSerialTransition := bSerialTransition AND gvl.remoteControls[nCounter]^.Execute(eCylinderCommands.COMMAND_A);
			END_IF
		END_FOR
		//Vacuum break , clean the air path
		IF bSerialTransition THEN
			//activate brakers
			THIS^.ActivateBreakers();
		END_IF
	eSpecialStates.INITIAL_STATE_2:
		bSerialTransition := timerBreak.Q;
		IF bSerialTransition THEN
			timerBreak.IN := FALSE;
			THIS^.InactivateBreakers();
		END_IF
	//-----------------------------
	//	Then check is vacuum jammed
	//-----------------------------
	eSpecialStates.INITIAL_STATE_3:
		bSerialTransition:=TRUE;
		THIS^.TurnVerifyVacuums(eCylinderCommands.COMMAND_B);
	eSpecialStates.INITIAL_STATE_4:
		bSerialTransition:=timerBreak.Q AND_THEN THIS^.TurnVerifyVacuums(eCylinderCommands.COMMAND_B);
		IF timerBreak.Q AND_THEN (NOT THIS^.TurnVerifyVacuums(eCylinderCommands.COMMAND_B)) THEN
			THIS^.AlarmCode := ERR_VACUUM_JAMMED;
		END_IF	
		IF bSerialTransition THEN
			timerBreak.IN := FALSE;
			THIS^.TurnVerifyVacuums(eCylinderCommands.COMMAND_A);
		END_IF
	//------------
	//	MACHNICAL INITIALIZE : SCARA/RACK FIRST
	//------------	
	eSpecialStates.INITIAL_STATE_5:	
		bSerialTransition:=TRUE;
		FOR nCounter :=0 TO 1 BY 1 DO
			bSerialTransition := bSerialTransition AND  members[nCounter]^.Initialize();
		END_FOR
	eSpecialStates.INITIAL_STATE_6:
		//------------
		//	THEN INDEX (in case of collision of clampers
		//------------
		bSerialTransition:= members[2]^.Initialize();
		IF bSerialTransition THEN
			NextState:=eSpecialStates.INITIAL_END;
		END_IF
	//------------------------------------------
	// Initialize - Group start (base procedure)
	//------------------------------------------
	eSpecialStates.GENERIC_GROUP_START:
		FOR nCounter :=0 TO 2 BY 1 DO
			IF members[nCounter]<>0 THEN
				members[nCounter]^.NextState := eSpecialStates.GENERIC_GROUP_START;
			END_IF
		END_FOR
		THIS^.TurnRackIdleDetection(FALSE);
		
		
		bSerialTransition:=TRUE;
	eSpecialStates.GENERIC_GROUP_IDLE:
		//---------------------
		//	IDLE (Engineering mode): wait command / able to trigger individual process
		//---------------------
		IF commStartProductionMode THEN
			//---------------------------
			//	Production mode
			//  1. Execute SCARA ASSEMBLE
			//	2. When purge command raise , coordinate stations to stop
			//---------------------------
			clamper1^.bIsBypassed := FALSE;
			clamper2^.bIsBypassed := FALSE;
			
			scara1^.PropTask := eSCARATask.task_assemble_scara1;
			scara1^.isTaskEngaged := TRUE;
			scara2^.PropTask := eSCARATask.task_snap_scara2;
			scara2^.isTaskEngaged := TRUE;	
			
			bSerialTransition := TRUE;
		ELSIF commStartTrialAssemble THEN
			//---------------------------
			//	Trial-assemble mode
			//---------------------------
			clamper1^.bIsBypassed := FALSE;
			clamper2^.bIsBypassed := TRUE;
			
			scara1^.PropTask := eSCARATask.task_assemble_scara1;
			scara1^.isTaskEngaged := TRUE;
			
			scara2^.PropTask := eSCARATask.task_snap_scara2;
			scara2^.isTaskEngaged := TRUE;
			
			
			
			bSerialTransition := TRUE;
		ELSIF commStartTrialSnap THEN
			//---------------------------
			//	Trial-snap mode
			//---------------------------
			clamper1^.bIsBypassed := FALSE;
			clamper2^.bIsBypassed := FALSE;
			bridge1^.bIsBypassed := TRUE;
			
			scara1^.isTaskEngaged := FALSE;
			
			scara2^.PropTask := eSCARATask.task_snap_scara2;
			scara2^.isTaskEngaged := TRUE;
			
			
			bSerialTransition := gvl.cylinderControls[Cy16].Execute(eCylinderCommands.COMMAND_B);
		ELSIF commStartRegularCheckMode THEN
			NextState := 16#300;
		END_IF
		
		IF bSerialTransition THEN
			
			THIS^.TurnDryRun(commIsDryRun); //activate dry run
			
			IF commStartTrialAssemble THEN
				gvl.cylinderControls[Cy6].isShutVerification := TRUE;
			END_IF
			IF commStartTrialSnap THEN	
				//--------------
				//	Turn off AOI
				//--------------
				aoi^.bIsBypassed := TRUE;
			END_IF
			
			THIS^.TurnRackIdleDetection(TRUE);
			//-------------------
			//speed factor renew
			//-------------------
			scara1^.context_out_speedFactor := commSpeedFactor;
			scara2^.context_out_speedFactor := commSpeedFactor;
		
			NextState := 16#1000;
		END_IF
		
		loader^.isWorking := bSerialTransition; //activate loader vacuum
		
	//------------------------
	//Working
	//------------------------
	16#300:
		//----------------------------------
		//	Regular check mode
		//	1. Stand-along check SCARA1/SCARA2
		//	1. Bypass some stations then feed-in parts in Slot1 , then transit to AOI
		//  2. Prompt meesage/door interlock
		//----------------------------------
		scara1^.isTaskEngaged := TRUE;
		
		clamper1^.bIsBypassed := TRUE;
		clamper2^.bIsBypassed := TRUE;
		
		bSerialTransition := TRUE;
	16#301:
		bSerialTransition := NOT scara1^.isTaskEngaged;
		IF bSerialTransition THEN
			scara2^.isTaskEngaged := TRUE;
		END_IF
	16#302:
		bSerialTransition := NOT scara2^.isTaskEngaged;
		IF bSerialTransition THEN
			commStartRegularCheckMode := false;
		END_IF
		//------------------------
		//AOI shuffing test
		//------------------------
	
		//---------------------------
		//	Purging chain
		//---------------------------
	16#1000:
		bSerialTransition := isPurged; //would be triggered by interfaceControl
	16#1001:
		bSerialTransition := scara2^.context_in_purgeack2.0;
		IF bSerialTransition THEN
			THIS^.isPurged := FALSE; //going to reset
		END_IF
	16#1002:
		bSerialTransition := NOT scara2^.context_in_purgeack2.0 ;
		IF bSerialTransition THEN
			FOR nCounter:=0 TO 3 BY 1 DO
				racks[nCounter]^.commEject := TRUE; //eject
			END_FOR	
		
			commStartProductionMode := FALSE;
			commStartTrialAssemble:= FALSE;
			commStartTrialSnap :=FALSE;
			
			NextState := eSpecialStates.GENERIC_GROUP_IDLE;
		END_IF		
	
END_CASE

ACTION ActivateBreakers:
backSecureBreaker := TRUE;
filterBreaker := TRUE;
timerBreak.IN := TRUE;
END_ACTION

ACTION InactivateBreakers:
backSecureBreaker := FALSE;
filterBreaker := FALSE;
timerBreak.IN := false;
END_ACTION

METHOD TurnDryRun : BOOL
VAR_INPUT
	isEnabled : bool;
END_VAR
//---------------------------------------------------
//turn off following devices if dry run	(no products)
//---------------------------------------------------
FOR nCounter:=0 TO 7 DO
	IF dryRunDevicesList[nCounter]<>0 THEN
		dryRunDevicesList[nCounter]^.isShutVerification := isEnabled;
	END_IF	
END_FOR
loader^.isSlotValidOverride := isEnabled;
aoi^.bIsBypassed := isEnabled;
scara1^.context_out_isDryRun.0 := isEnabled;
scara2^.context_out_isDryRun.0 := isEnabled;
IF isEnabled THEN
	gvl.cylinderControls[Cy16].Execute(eCylinderCommands.COMMAND_B);
END_IF
END_METHOD

METHOD TurnRackIdleDetection : BOOL
VAR_INPUT
	value : bool;
END_VAR
FOR nCounter:=0 TO 3 BY 1 DO
	IF racks[nCounter] <>0 THEN
		racks[nCounter]^.isIdleDetection := value;
	END_IF		
END_FOR
END_METHOD

METHOD TurnVerifyVacuums : BOOL
VAR_INPUT
	command : eCylinderCommands;
END_VAR
TurnVerifyVacuums := TRUE; //return , true : none of vacuum generated,  false : any of vacuum generated
FOR nCounter:=0 TO 6 BY 1 DO
	IF gvl.verifyVacuums[nCounter]<>0 THEN
		TurnVerifyVacuums := TurnVerifyVacuums AND NOT gvl.verifyVacuums[nCounter]^.Execute(command);
	END_IF	
END_FOR

CASE command OF
	eCylinderCommands.COMMAND_B:
		timerBreak.IN := TRUE;
	eCylinderCommands.COMMAND_A:
		timerBreak.IN := FALSE;
END_CASE
END_METHOD

END_FUNCTION_BLOCK

// ---- POUs/Stations/HRASI/RunScaraAgent.TcPOU
FUNCTION_BLOCK RunScaraAgent EXTENDS RunUnitGeneric
VAR_INPUT
	isTaskEngaged : BOOL;		//triggered by coordinator , reset by myself
	//-------------------
	// Remote control - Input
	//-------------------
	out_start_0 AT %Q* : BIT;
	out_selProg1_1 AT%Q* : BIT;
	out_selProg2_2 AT%Q* : BIT;
	out_selProg4_3 AT%Q* : BIT;
	
	out_stop_4 AT%Q* :BIT; //foced stop, not recommend to use
	
	out_pause_5 AT%Q* : BIT;		
	out_continue_6 AT%Q* : BIT;
	
	out_reset_7 AT%Q* : BIT; 	//error reset
	//------------------
	//	CONTEXT 
	//------------------
	context_out_alarmAck AT%Q* : WORD;
	context_out_perNodePurged2 AT%Q* : BYTE;	// the purge request
	context_out_productType AT%Q* : BYTE;
	context_out_isSlotValid AT%Q* : BYTE;
	context_out_perNodePurged1 AT%Q* : BYTE;
	context_out_speedFactor AT%Q* : BYTE; // in percentage
	context_out_isDryRun AT%Q* : BYTE;
END_VAR
VAR_OUTPUT
	//-------------------
	// Remote control - Output
	//-------------------
	in_ready_0 AT%I* : BIT; //Turns ON when the controller startup completes and no task is running. 
	in_running_1 AT%I* : BIT; //Turns ON when task is running. However, turns OFF when “Paused output” is ON. 
	in_paused_2 AT%I* : BIT; //
	in_error_3 AT%I* : BIT;
	in_eStop_4 AT%I* : BIT;		//as EDM
	in_safeGuard_5 AT%I* : BIT;	//as EDM to safeguard
	in_sError_6 AT%I* : BIT;
	in_warning_7 AT%I* : BIT;
	//------------------
	//	CONTEXT 
	//------------------
	context_in_alarmCode AT%I* : WORD;
	context_in_purgeack1 AT%I* : BYTE;
	context_in_purgeack2 AT%I* : BYTE;
	
	context_in_taskState AT%I* : BYTE;
	context_in_setSlotValid AT%I* : BYTE;
	
END_VAR
VAR CONSTANT
	taskInit : UINT := 1;
	taskAssembly : UINT :=2;
	taskSnipFit : UINT :=3;
	taskRegularCheck : UINT :=3;
	
	taskEngCalibration : UINT :=4;
	taskEngPickAndDrip : UINT:=5;
END_VAR
VAR PERSISTENT
	timer : TON;
END_VAR

//mission:
//2. sequence start/stop as Remote I/O

//Select Program first then Start
//Stop program

//Pause program
//Continue when ready on

SUPER^();
timer();

//transmit purged status
context_out_perNodePurged1.0 := (previousNode<>0 AND_THEN previousNode^.isPurged);
context_out_isSlotValid.0 := SlotLast<>0 AND_THEN SlotLast^.Valid;
isPurged := context_in_purgeack1.0 ;// reflect purge ack status

//----------------------
//	Task running control
//----------------------
IF bPause AND NOT in_paused_2 AND in_running_1 THEN
	out_pause_5 := TRUE;
	out_continue_6 := FALSE;
ELSIF NOT bPause AND in_paused_2  THEN
	out_pause_5 := FALSE;
	out_continue_6 := TRUE;
ELSE
	out_pause_5 := FALSE;
	out_continue_6 := FALSE;
END_IF

IF timer.Q THEN
	timer.IN := FALSE;
	out_reset_7 := FALSE;
	out_stop_4 := FALSE;
	context_out_alarmAck:=0;
END_IF

CASE outputState OF 	
	eSpecialStates.INITIAL_BEGIN:	
		isTaskEngaged := FALSE;
		out_start_0 := FALSE;
		out_stop_4 := TRUE;
		bSerialTransition := TRUE;
	//----------------
	//Check no running
	//----------------		
	eSpecialStates.INITIAL_STATE_1:
		bSerialTransition := NOT in_running_1 AND in_ready_0;
		IF bSerialTransition THEN
			//initializing process activated
			PropTask := eSCARATask.task_init;
			
			out_stop_4 := FALSE; //release
			
			// Forced reset error
			THIS^.ErrorClear(eErrorClearWays.RESET);
		END_IF
	//-------------------
	// Forced reset error done
	//-------------------
	eSpecialStates.INITIAL_STATE_2:
		bSerialTransition := NOT out_reset_7; 
	//--------------
	//Check no error and ready
	//--------------
	eSpecialStates.INITIAL_STATE_3:
		bSerialTransition := (NOT in_error_3) AND NOT in_running_1 AND in_ready_0;
		IF bSerialTransition THEN
			out_start_0 := TRUE;		
		END_IF
	//Start initializing , Check running
	eSpecialStates.INITIAL_STATE_4:
		bSerialTransition := in_running_1 AND NOT in_ready_0;
		IF bSerialTransition THEN
			out_start_0 := FALSE; //after process started , pause
		END_IF
	//Start initializing, Check ran
	eSpecialStates.INITIAL_STATE_5:
		bSerialTransition := NOT in_running_1 AND  in_ready_0;
		IF bSerialTransition THEN
			out_start_0 := FALSE;
			NextState := eSpecialStates.INITIAL_END;
		END_IF
	//-------------------------------
	// IDLE/Program selection states.
	//------------------------------
	eSpecialStates.GENERIC_GROUP_START:
		//--------------
		// Program selected and triggered
		//--------------
		bSerialTransition := isTaskEngaged;
	16#1:
		bSerialTransition := NOT in_running_1 AND  in_ready_0;
		IF bSerialTransition THEN
			out_start_0 := TRUE;
		END_IF
		
	16#2:
		bSerialTransition := in_running_1 AND NOT in_ready_0;
		IF bSerialTransition THEN
			out_start_0 := FALSE;
			NextState := 16#200;
		END_IF
		//------------------------------------------------------------------
		// Operating
		//------------------------------------------------------------------
	16#200:
		//task finished natually or request purge from previous node
		bSerialTransition := NOT in_running_1 AND in_ready_0;
		IF bSerialTransition THEN
			//succesfully stopped
			isTaskEngaged := FALSE;
			NextState := eSpecialStates.GENERIC_GROUP_START;
		END_IF	
END_CASE

METHOD ConfigureRead : CellDataBlock
VAR_INPUT
	input : CellDataBlock; //would offer sub-index ...etc
	mode : eModes;
END_VAR
END_METHOD

METHOD ConfigureWrite : BOOL
VAR_INPUT
	input : CellDataBlock;
	mode : eModes;
END_VAR
//Implemented by concre derived class
ConfigureWrite := true;
END_METHOD

METHOD Control : BOOL
VAR_INPUT
	input : CellDataBlock;
	mode : eModes; //commit mode
END_VAR
bEnStep := input.unit.base.controlWord.bit0EnStep;
bTrigStep := input.unit.base.controlWord.bit1TrigStep;
bPause := input.unit.base.controlWord.bit2StatePause;
bIsBypassed := input.unit.base.controlWord.bit3IsBypassed;
bWorkingOverride := input.unit.base.controlWord.bit4WorkingOverride;
bMaterialOverride := input.unit.base.controlWord.bit5MaterialOverride;
Control:=true;
END_METHOD

METHOD ErrorClear : BOOL
VAR_INPUT
	input : eErrorClearWays;
END_VAR
//context_out_alarmAck := 0; // ack reset
out_reset_7 := TRUE;
context_out_alarmAck := 1;

timer.IN := TRUE; //activate  timer

IF in_eStop_4 THEN
	out_stop_4 := true; //addtionally make sure procedure stopped
END_IF
END_METHOD

METHOD ErrorDetect : UDINT
VAR_INPUT
END_VAR


IF in_eStop_4 THEN

	ErrorDetect := eErrorReasons.ERR_EMG;
ELSIF in_safeGuard_5 THEN
	ErrorDetect := eErrorReasons.ERR_SAFETY;
	
ELSIF in_error_3 OR context_in_alarmCode<>0 THEN
	IF context_in_alarmCode = 0 THEN
		ErrorDetect := eErrorReasons.ERR_GENERIC_ERROR; //default unknown alarm
	ELSE
		ErrorDetect := context_in_alarmCode; //user defined error code
	END_IF
ELSE
	//Healthy , no error
	ErrorDetect := 0;
END_IF
END_METHOD

METHOD Monitor : CellDataBlock
VAR_INPUT
END_VAR
Monitor.unit.base.controlWord.bit0EnStep := bEnStep;
Monitor.unit.base.controlWord.bit1TrigStep := bTrigStep;
Monitor.unit.base.controlWord.bit2StatePause := bPause;
Monitor.unit.base.controlWord.bit3IsBypassed := bIsBypassed;
Monitor.unit.base.controlWord.bit4WorkingOverride := bWorkingOverride;
Monitor.unit.base.controlWord.bit5MaterialOverride := bMaterialOverride;
//Transition status
Monitor.unit.base.transitionByte := transitionByte;
//
Monitor.unit.base.alarmCode := TO_WORD(AlarmCode);

//reflect task state instead
Monitor.unit.base.state := TO_WORD(THIS^.context_in_taskState);
Monitor.unit.base.nextState := TO_WORD(THIS^.context_in_taskState);

//
IF workingTimer.IN THEN
	//timer is running , reflect real value
	Monitor.unit.base.workingTimerCache := TO_DWORD(workingTimer.ET);
ELSE
	//timer is stopped , reflect cached value
	Monitor.unit.base.workingTimerCache := TO_DWORD(workingTimerCache);
END_IF
END_METHOD

PROPERTY PUBLIC PropTask : eSCARATask
GET

PropTask.0 := out_selProg1_1;
PropTask.1 := out_selProg2_2;
PropTask.2 := out_selProg4_3;
END_GET
SET
out_selProg1_1 := ((PropTask AND 16#01) > 0);
out_selProg2_2 := ((PropTask AND 16#02) > 0);
out_selProg4_3 := ((PropTask AND 16#04) > 0);
END_SET
END_PROPERTY

METHOD TypeCode : eCategrories
VAR_INPUT
END_VAR
TypeCode := eCategrories.SELECTION_UNIT;
END_METHOD

END_FUNCTION_BLOCK

// ---- POUs/Stations/HRASI/RunClamper.TcPOU
FUNCTION_BLOCK RunClamper EXTENDS RunUnitSlave
VAR_INPUT
END_VAR
VAR_OUTPUT
END_VAR
VAR
	//devices
	horizon : POINTER TO RunCylinder;
	clamper : POINTER TO RunCylinder;
	//
	configSnap : BOOL; //set true for instance of Snap
	
	//
	tickTime AT%Q*: DWORD ; //in ms
	commIdTrigger AT%Q* : DWORD;
	
	//
	alignCounter : INT;
END_VAR
VAR CONSTANT
	bScaraReady : INT := 1;
END_VAR
VAR PERSISTENT
	alignIteration : INT := 0;
END_VAR

SUPER^();

//Link to :
// 1. Indexer - working signal
// 2. Bridge - working signal dispatch  to SCARA

tickTime := TIME_TO_DWORD(workingTimerCache);

CASE outputState OF
	//---------------------------
	//	Initialization : hold and push
	//---------------------------	
	eSpecialStates.INITIAL_BEGIN:
		clamper^.isRemoteControl := FALSE; //off remote control
		bSerialTransition := clamper^.Execute(eCylinderCommands.NO_COMMAND); //remain
	eSpecialStates.INITIAL_STATE_1:
		bSerialTransition := horizon^.Execute(eCylinderCommands.COMMAND_B);
	eSpecialStates.INITIAL_STATE_2:
		bSerialTransition := clamper^.Execute(eCylinderCommands.COMMAND_A); //release
	eSpecialStates.INITIAL_STATE_3:
		bSerialTransition := horizon^.Execute(eCylinderCommands.COMMAND_A); //back
	eSpecialStates.INITIAL_STATE_4:
		bSerialTransition := TRUE;
	eSpecialStates.INITIAL_STATE_5:
		bSerialTransition := TRUE;
		IF bSerialTransition THEN
			NextState := eSpecialStates.INITIAL_END;
		END_IF
	//----------------------------
	//	Working
	//----------------------------
	eSpecialStates.SLAVE_ENTER_PROCEDURE:
		IF bMaterialOverride THEN
			alignCounter := 0; //reset
			bSerialTransition := TRUE;
		ELSE
			NextState := 16#207; //bypass
		END_IF
	16#201:
		//Indexer in position , horizonin
		bSerialTransition := horizon^.Execute(eCylinderCommands.COMMAND_B) AND clamper^.Execute(eCylinderCommands.COMMAND_A);
	16#202:
		transitionByte.0 := clamper^.Execute(eCylinderCommands.COMMAND_B);
		transitionByte.1 := alignCounter >= alignIteration;
		
		IF transitionByte = 1 THEN
			alignCounter := alignCounter+1;
			NextState := 16#201; // realign
		ELSIF transitionByte = 3 THEN
			 bSerialTransition := TRUE ; // go ahead
		ELSE
			// clamper mechanical movement
		END_IF
	
	16#203:
		transitionByte.0 := horizon^.Execute(eCylinderCommands.COMMAND_A);
		transitionByte.1 := TRUE;
		
		IF transitionByte = 16#3 THEN
			
			slaveWorkingSignal[bScaraReady]:= TRUE; //trigger SCARA agent
			
			IF configSnap THEN
				clamper^.isRemoteControl := TRUE; // gave scara remote control
			END_IF
			
			bSerialTransition := TRUE;
		END_IF
	16#204:
		//Wait SCARA 
		bSerialTransition := NOT slaveWorkingSignal[bScaraReady];
		IF bSerialTransition AND previousNode<>0 AND_THEN previousNode^.isPurged  THEN
			isPurged := TRUE; //no further part would coming
		END_IF
		IF bSerialTransition THEN
			clamper^.isRemoteControl := FALSE; // demolish remote control
			commIdTrigger := SlotBase^.Id; //trigger the data logger
		END_IF
	16#205:
		//send part back to indexer
		bSerialTransition := clamper^.Execute(eCylinderCommands.COMMAND_B);
	16#206:
		//send part back to indexer
		bSerialTransition := horizon^.Execute(eCylinderCommands.COMMAND_B);
	16#207:
		//release part 
		bSerialTransition := clamper^.Execute(eCylinderCommands.COMMAND_A); //release
	16#208:
		//empty clamper extract
		IF horizon^.Execute(eCylinderCommands.COMMAND_A) THEN
			NextState := eSpecialStates.SLAVE_WORK_DONE;
		END_IF
	
	//-------------
	//	Last station should treated as empty
	//-------------
	eSpecialStates.SLAVE_WORK_DONE:
		// auto reset last slot
		IF configSnap THEN
			SlotBase^.Valid := FALSE;
		END_IF
		
		//bypass purge status
		IF NOT SlotBase^.Valid AND previousNode<>0 AND_THEN previousNode^.isPurged THEN
			isPurged := TRUE;
		END_IF
		
END_CASE

METHOD FB_init : BOOL
VAR_INPUT
	bInitRetains : BOOL; // if TRUE, the retain variables are initialized (warm start / cold start)
	bInCopyCode : BOOL;  // if TRUE, the instance afterwards gets moved into the copy code (online change)
	
	argParent : POINTER TO RunUnitGeneric;
	argSlotBase : POINTER TO RunMaterial;
	argSlotLast : POINTER TO RunMaterial;
	
	argWorkingSignal : POINTER TO BOOL;
	
	argHorizon : POINTER TO RunCylinder;
	argClamper : POINTER TO RunCylinder;
	argConfigSnap : BOOL;
END_VAR
//initialize 
Parent := argParent;
SlotBase := argSlotBase;
SlotLast := argSlotLast;
//
IF bInitRetains THEN
	NextState := eSpecialStates.INITIAL_BEGIN;
END_IF

workingSignal := argWorkingSignal; //link

//device link
horizon := argHorizon;
clamper := argClamper;
configSnap := argConfigSnap;
END_METHOD

END_FUNCTION_BLOCK

// ---- POUs/Stations/HRASI/RunLoading.TcPOU
FUNCTION_BLOCK RunLoading EXTENDS RunUnitSlave
VAR_INPUT
	externalSlotValid  : BOOL;
	isSlotValidOverride AT%M* : BOOL; //eniginnering use , dry run
	isWorking : bool;
	
	refSensorPairs : POINTER TO ARRAY[0..3] OF defSensorPair; //define stations sensor flag signatures
	refFixtures : pointer to helperOutputSelection;
END_VAR
VAR_OUTPUT
	//purgeRequest AT%Q* : BOOL; //link to SCARA2
END_VAR
VAR	
	existence : POINTER TO RunSignal;	
	//watchDog : TON;
	
	totalCount AT%M* : UDINT; 
END_VAR
VAR PERSISTENT
	currentId : DWORD;
END_VAR

SUPER^();

//-------------------------------
//	Slot-1 to loading bottom part
//-------------------------------
CASE outputState OF
	eSpecialStates.INITIAL_BEGIN:
//		purgeRequest := FALSE;
		NextState := eSpecialStates.INITIAL_END;
	//---------------------
	//	Working
	//---------------------
	eSpecialStates.SLAVE_ENTER_PROCEDURE:
		//check if empty
		bSerialTransition := existence^.debouncedOff;
		IF bSerialTransition THEN
			
			SlotBase^.Valid := FALSE; //always false in beginning
			slaveWorkingSignal[1] := TRUE; // trigger scara to put
					
		ELSIF existence^.debouncedOn THEN
			THIS^.AlarmCode := eErrorReasons.ERR_PART_MISSING;
		END_IF
	16#201:
		bSerialTransition := NOT slaveWorkingSignal[1]; //scara should set valid before reset working 
		IF bSerialTransition THEN
			//Off back secure
			IF refFixtures <> 0 THEN
				refFixtures^.Trigger(refSensorPairs^[0],FALSE); 
			END_IF
			SlotBase^.Valid := externalSlotValid OR isSlotValidOverride ; //transit
		ELSE
			//Activate back secure
			IF refFixtures <> 0 THEN
				refFixtures^.Trigger(refSensorPairs^[0],isWorking); 
			END_IF
		END_IF
	16#202:
		//check if material status matched sensor status
		bSerialTransition := (SlotBase^.Valid = existence^.debouncedOn) OR isSlotValidOverride;
		
		IF bSerialTransition AND (previousNode<>0 AND_THEN previousNode^.isPurged) AND NOT SlotBase^.Valid THEN
			isPurged := TRUE;
			
		ELSIF (NOT isSlotValidOverride) AND   SlotBase^.Valid AND existence^.debouncedOff  THEN
			AlarmCode := eErrorReasons.ERR_PART_MISSING; // absense
		ELSIF (NOT isSlotValidOverride) AND (NOT SlotBase^.Valid  AND existence^.debouncedOn)  THEN
			AlarmCode := eErrorReasons.ERR_PART_REMAINED; // abnormal
		END_IF
				
		IF bSerialTransition AND SlotBase^.Valid THEN
			//give material id
			SlotBase^.Id := currentId;
			currentId := IncNoOverflow(input:= currentId);
			totalCount := IncNoOverflow(input:= totalCount); //bottom part inlet count
		END_IF
		
	16#203:
		NextState := eSpecialStates.SLAVE_WORK_DONE;
END_CASE

METHOD ErrorClear : BOOL
VAR_INPUT
	input : eErrorClearWays;
END_VAR
IF AlarmCode = eErrorReasons.ERR_PART_MISSING THEN
	SlotBase^.Valid := false; //just let it go
END_IF
AlarmCode := 0; //code reset to 0
timeoutTimer.IN := FALSE; //reset
END_METHOD

METHOD FB_init : BOOL
VAR_INPUT
	bInitRetains : BOOL; // if TRUE, the retain variables are initialized (warm start / cold start)
	bInCopyCode : BOOL;  // if TRUE, the instance afterwards gets moved into the copy code (online change)
	
	argParent : POINTER TO RunUnitGeneric;
	argSlotBase : POINTER TO RunMaterial;
	argSlotLast : POINTER TO RunMaterial;
	
	argWorkingSignal : POINTER TO BOOL;
	
	argExistence : POINTER TO RunSignal;
END_VAR
//initialize 
Parent := argParent;
SlotBase := argSlotBase;
SlotLast := argSlotLast;
//
IF bInitRetains THEN
	NextState := eSpecialStates.INITIAL_BEGIN;
END_IF

workingSignal := argWorkingSignal; //link

existence := argExistence;
END_METHOD

END_FUNCTION_BLOCK

// ---- POUs/Stations/HRASI/helperOutputSelection.TcPOU
FUNCTION_BLOCK helperOutputSelection
VAR_INPUT
END_VAR
VAR_OUTPUT
END_VAR
VAR
	outputs AT%Q*: ARRAY[0..3] OF BOOL;
	
	nCounter : INT;
END_VAR

ACTION ReleaseAll:
FOR nCounter:=0 TO 3 BY 1 DO
	outputs[nCounter] := false;
END_FOR
END_ACTION

METHOD Trigger : BOOL
VAR_INPUT
	sensorPair : defSensorPair;
	state : BOOL; //ON/OFF
END_VAR
VAR
	index : BYTE;
END_VAR
index.0 := sensorPair.bit0;
index.1 := sensorPair.bit1;

outputs[index] := state;
END_METHOD

END_FUNCTION_BLOCK

// ---- POUs/Stations/HRASI/RunAoiInspectionV1.TcPOU
FUNCTION_BLOCK RunAoiInspectionV1 EXTENDS RunUnitSlave
VAR_INPUT
	ngBinReady : BOOL;
	ngCounter : POINTER TO UDINT;
	
	productType : BYTE; // input , 0:S 1:V 2: BGSx
	
	statusCoaxial : BYTE;
	statusStripper : BYTE;
	
END_VAR
VAR_OUTPUT
	commandCoaxial : BYTE;
	commandStripper : BYTE;
END_VAR
VAR
	//devices
	ngCylinder : POINTER TO RunCylinder; // normal close cylinder
	
	aoiOut1Done AT%I* : BOOL ; //done , if error comes , this line wont be on
	aoiOut2Grade AT%I* : BOOL ; //ok/ng
	
	aoiTrigger AT%Q* : BOOL;	
	aoiOnline AT%M* : BOOL;
	aoiBGSxEnable AT%Q* : BOOL; // 1: enable BGSx inspection , 0: disenable as regular V-Top
	//internal
	
	commIdTrigger AT%Q* : DWORD;
	
	aoiTimeoutTimer : ton;
	aoiSwitchingTimer : ton;
	aoiOverallGrade : BOOL;
	//
	serialNGCounter : INT;
	
	//
	currentCheck : INT := CHECK_REGULAR;
	targetCheck : INT := CHECK_BGSx;
END_VAR
VAR PERSISTENT
	serialNGGoal AT%M* : INT ;
	
	intensityCoaxial AT%M* : BYTE := 0;
	intensityStrip AT%M* : BYTE := 0;
END_VAR
VAR CONSTANT
	CHECK_REGULAR : INT := 0;
	CHECK_BGSx : INT :=1;
END_VAR

SUPER^();

//----------------
//	AOI OFFLINE 
//-----------------
timeouttimer.IN := (NOT  aoiOnline);
IF timeouttimer.Q AND NOT aoiOnline THEN
	AlarmCode:= eErrorReasons.ERR_OFFLINE;
END_IF
aoiTimeoutTimer(PT:= T#30S);
aoiSwitchingTimer(pt :=T#100MS);

CASE outputState OF
	//--------------------------------
	//	Initialization TODO, (Light on?)
	//--------------------------------	
	eSpecialStates.INITIAL_BEGIN:	
		bSerialTransition := ngCylinder^.Execute(eCylinderCommands.COMMAND_A);
		IF bSerialTransition THEN
			serialNGCounter := 0;
			aoiTrigger := FALSE;
		END_IF
	eSpecialStates.INITIAL_STATE_1:
		bSerialTransition := NOT aoiOut1Done;
		IF bSerialTransition THEN
			NextState := eSpecialStates.INITIAL_END;
		END_IF
	//---------------------------------
	//	Working
	//---------------------------------
	eSpecialStates.SLAVE_ENTER_PROCEDURE:
		// report id to SCADA?		
		transitionByte.0 := ngCylinder^.Execute(eCylinderCommands.COMMAND_A); //alway extend
		transitionByte.1 := NOT aoiOut1Done; //check aoi-done off
		
		bSerialTransition:= (transitionByte = 16#3);
		IF bSerialTransition THEN
			atomicOperation := TRUE;
			aoiOverallGrade := TRUE; //preset
			
			currentCheck := CHECK_REGULAR; //reset
			targetCheck  := CHECK_REGULAR;
			IF productType = 2 THEN
				targetCheck := CHECK_BGSx;
			END_IF
			
			IF NOT bMaterialOverride THEN
				NextState := 16#230; //no material , leave	
			END_IF
		ELSE
			//--------------------------
			//await mechanism switching	
			//--------------------------
		END_IF
	
	//--------------------------------
	//	Cyclic Trigger-Get Result : Start
	//--------------------------------
	16#201:
		IF NOT aoiSwitchingTimer.IN THEN
			aoiSwitchingTimer.IN := TRUE;
		END_IF
		
	
		CASE currentCheck OF
			CHECK_REGULAR :
				aoiBGSxEnable := FALSE;
				bSerialTransition := THIS^.switchDimmer(TRUE,FALSE) AND aoiSwitchingTimer.Q; // turn coaxial on , strip off
			CHECK_BGSx :
				aoiBGSxEnable := TRUE;
				bSerialTransition := THIS^.switchDimmer(FALSE,TRUE) AND aoiSwitchingTimer.Q; // turn coaxial off , strip on
		END_CASE
	
		IF bSerialTransition THEN
			aoiTrigger := TRUE; //set aoi-trigger on
			aoiTimeoutTimer.IN := TRUE;
			aoiSwitchingTimer.IN := FALSE; //reset for re-enter
		ELSE
			//await dimmer switching
		END_IF
		
	16#202:
		bSerialTransition := aoiOut1Done OR aoiTimeoutTimer.Q;
		IF aoiTimeoutTimer.Q THEN
			AlarmCode := eErrorReasons.ERR_PART_MISSING;
			aoiOverallGrade := FALSE; // once timeout , should be set as NG to be safe
		END_IF
		IF bSerialTransition THEN
			aoiTrigger := FALSE; //reset
		END_IF
	16#203:
		bSerialTransition := NOT aoiOut1Done;
		IF bSerialTransition THEN 
			
			aoiTimeoutTimer.IN := FALSE; //reset
			aoiOverallGrade := aoiOverallGrade AND aoiOut2Grade; // inclusive
			
			IF currentCheck = targetCheck THEN
				atomicOperation := FALSE;
				nextstate := 16#220;			  // conclude and output
			ELSE
				currentCheck := currentCheck +1 ; // do next check
				nextstate := 16#201;
			END_IF
		END_IF
	//--------------------------------
	//	Cyclic Trigger-Get Result : End
	//--------------------------------
	
	
		//-------------------------
		//	Output
		//-------------------------
	16#220:
		IF commIdTrigger <> SlotBase^.Id THEN
			commIdTrigger := SlotBase^.Id; //trigger the data logger
		END_IF
		
		//--------------------------
		//	OK : open gate
		//	NG : await until NG bin ready
		//--------------------------
		bSerialTransition := (aoiOverallGrade AND_THEN ngCylinder^.Execute(eCylinderCommands.COMMAND_B)) 
							OR ( (NOT aoiOverallGrade) AND_THEN ngBinReady);
		
		IF bSerialTransition THEN
			nextstate := 16#230;
			
			//-------------------------
			//	Data handling and warning
			//-------------------------
			IF aoiOverallGrade THEN
				serialNGCounter := 0; //reset
			ELSE
				SlotBase^.Valid := FALSE; //set as inexsited	
				serialNGCounter := serialNGCounter+1;
				IF  serialNGCounter >=  serialNGGoal THEN
					AlarmCode := eErrorReasons.ERR_CONSECUTIVE_NG;
					serialNGCounter := 0; //reset
				END_IF
				
				IF ngCounter<>0 THEN
					ngCounter^ := ngCounter^ +1; //count-up NG bin counter
				END_IF		
			END_IF
		ELSE
			//await machansim working
		END_IF
		//-------------------------
		// Task closed
		//------------------------	
	16#230:
			
		IF NOT SlotBase^.Valid AND previousNode <>0 AND_THEN previousNode^.isPurged THEN
			isPurged := true; // i am purged
		END_IF
			
		NextState := eSpecialStates.SLAVE_WORK_DONE;
END_CASE

METHOD FB_init : BOOL
VAR_INPUT
	bInitRetains : BOOL; // if TRUE, the retain variables are initialized (warm start / cold start)
	bInCopyCode : BOOL;  // if TRUE, the instance afterwards gets moved into the copy code (online change)
	
	argParent : POINTER TO RunUnitGeneric;
	argSlotBase : POINTER TO RunMaterial;
	argSlotLast : POINTER TO RunMaterial;
	
	argWorkingSignal : POINTER TO BOOL;
	
	argNgCylinder : POINTER TO RunCylinder;
	
END_VAR
//initialize 
Parent := argParent;
SlotBase := argSlotBase;
SlotLast := argSlotLast;
//
IF bInitRetains THEN
	NextState := eSpecialStates.INITIAL_BEGIN;
END_IF

workingSignal := argWorkingSignal; //link

ngCylinder := argNgCylinder;
END_METHOD

METHOD switchDimmer : BOOL
VAR_INPUT
	enableCoaxial : BOOL;
	enableStrip : BOOL;
END_VAR
IF enableCoaxial THEN
	commandCoaxial := intensityCoaxial;
ELSE
	commandCoaxial := 0;
END_IF

IF enableStrip THEN
	commandStripper := intensityStrip;
ELSE
	commandStripper := 0;
END_IF


//when status matched command means matched
switchDimmer := (commandCoaxial = statusCoaxial) AND (commandStripper = statusStripper);
END_METHOD

END_FUNCTION_BLOCK

// ---- POUs/Stations/HRASI/RunBridge.TcPOU
FUNCTION_BLOCK RunBridge EXTENDS RunUnitSlave
VAR_INPUT
	fakeAck AT%M* : BOOL;
END_VAR
VAR_OUTPUT
END_VAR
VAR
	bridge : defHandshake;
END_VAR

//----------------------------------------------
//	Bridge working signal and handshaking signal
//----------------------------------------------
SUPER^();

CASE outputState OF 
	//--------------------------------
	//	Initialization
	//--------------------------------	
	eSpecialStates.INITIAL_BEGIN:
		bridge.ready := FALSE;
		fakeAck:=FALSE;
		bSerialTransition := NOT bridge.ack AND NOT bridge.valid;
		IF bSerialTransition THEN
			NextState := eSpecialStates.INITIAL_END;
		END_IF
	//---------------------------------
	//	Working
	//---------------------------------
	eSpecialStates.SLAVE_ENTER_PROCEDURE:
		bridge.ready := TRUE;
		bSerialTransition := TRUE;
	16#201:
		bSerialTransition := bridge.ack OR fakeAck;
		IF bSerialTransition THEN
			fakeAck := FALSE; //auto-reset
			bridge.ready := FALSE;
		END_IF
	16#202:
		IF NOT bridge.ack THEN
			NextState := eSpecialStates.SLAVE_WORK_DONE;
		END_IF
END_CASE

END_FUNCTION_BLOCK

// ---- POUs/Stations/HRASI/RunCommonRack.TcPOU
FUNCTION_BLOCK RunCommonRack EXTENDS RunUnitGeneric
VAR_INPUT
	//isEject : BOOL; //link to coordinator
	commEject AT%M* : BOOL; // link to HMI
	isIdleDetection : BOOL;
END_VAR
VAR_OUTPUT
END_VAR
VAR
	
	button : POINTER TO RunSignal ;
	fixer : POINTER TO RunCylinder;
	approx : POINTER TO RunSignal; // approx then lock
	
	signal : ProgrammedOutput;
	//---------------------------------
	//	Over Fieldbus linked with SCARA
	//---------------------------------
	rackReady AT%Q*: BOOL;
	rackEngaged AT%I*: BOOL;	

	items : ARRAY[0..5] OF defItem; // 5th material - Exceed Prefilter
	
	//---------------------------------
	//	Internal
	//---------------------------------
	nCounter : INT;
END_VAR
VAR_STAT PERSISTENT
	//F1,F2,F3,Bottom,Top,Excess filter
	// LCM(84,81,72) = 4536
	// LCM(84,81) = 2268
	// LCM(81,72) = 648  , 8 x F3/F2/F1 , 9 x EP , about 2 hours
	Bounds : ARRAY[0..5] OF BYTE := [84,88,81,40,40,72]; // 5th material - Exceed Prefilter
END_VAR


//Control the working flow of rack

SUPER^();
signal();

IF NOT rackReady AND NOT approx^.debouncedOn THEN
	signal.Activate(0);//100% set light flicking
ELSIF NOT rackReady AND  approx^.debouncedOn THEN
	signal.Activate(2);//25% flicking
ELSIF rackReady THEN
	signal.Deactivate();
END_IF

IF button^.onTimeElapsed > T#2S THEN
	commEject := TRUE;
END_IF

CASE outputState OF
	//----------------
	//	Initialization
	//----------------
	eSpecialStates.INITIAL_BEGIN:
		WarningCode := 0;
		NextState:=eSpecialStates.INITIAL_END;
	//-----------------
	//	Working
	//-----------------
	eSpecialStates.GENERIC_GROUP_START:
		//make sure all counter reseted by SCARA
		bSerialTransition := TRUE;
		FOR nCounter := 0 TO 4 DO
			bSerialTransition := bSerialTransition AND (items[nCounter].CurrerntIndex = 0);
		END_FOR
	16#1:
		//rack is empty
		rackReady := FALSE; //released
		commEject := FALSE;
		bSerialTransition := fixer^.Execute(eCylinderCommands.COMMAND_A)AND button^.debouncedOff; //relase
		
	16#2:
		bSerialTransition := approx^.debouncedOn AND button^.onTimeElapsed > T#100MS; //wait until rack closed
		IF approx^.debouncedOn THEN			
			timeouttimer.IN := TRUE;
		END_IF
		IF approx^.debouncedOn AND NOT bSerialTransition  AND timeouttimer.Q AND isIdleDetection THEN
			WarningCode := eErrorReasons.ERR_IDLE;
		END_IF
		IF bSerialTransition OR NOT approx^.debouncedOn  THEN
			WarningCode := 0;
			timeouttimer.IN := FALSE; //leave with reset
		END_IF
	16#3:
		bSerialTransition := fixer^.Execute(eCylinderCommands.COMMAND_B); //lock
		IF bSerialTransition THEN
			
			rackReady := TRUE;
		END_IF
	16#4:
		//------------------------------------------------------------------
		//	Check if any item reached the bound. then set rackReady as false
		// or by external signal (manual or job stop)
		//------------------------------------------------------------------
		FOR nCounter := 0 TO 5 DO
			IF items[nCounter].CurrerntIndex >= Bounds[nCounter] THEN
				bSerialTransition := TRUE;	
			END_IF
		END_FOR
		bSerialTransition := bSerialTransition OR  commEject ;
		
		IF bSerialTransition THEN
			rackReady := FALSE; //released
		END_IF
	16#5:
		//wait until SCARA disengaged
		IF NOT rackEngaged THEN
			NextState := eSpecialStates.GENERIC_GROUP_START; //rewind
		END_IF
END_CASE

METHOD FB_init : BOOL
VAR_INPUT
	bInitRetains : BOOL; // if TRUE, the retain variables are initialized (warm start / cold start)
	bInCopyCode : BOOL;  // if TRUE, the instance afterwards gets moved into the copy code (online change)
	
	argParent : POINTER TO RunUnitGeneric;
	argSlotBase : POINTER TO RunMaterial;
	argSlotLast : POINTER TO RunMaterial;
	
	argButton : POINTER TO RunSignal ;
	argFixer : POINTER TO RunCylinder;
	argApprox : POINTER TO RunSignal; 
END_VAR
//initialize 
Parent := argParent;
SlotBase := argSlotBase;
SlotLast := argSlotLast;
//
IF bInitRetains THEN
	NextState := eSpecialStates.INITIAL_BEGIN;
END_IF

IF Bounds[0] = 0 THEN
	//initialize bounds
	Bounds[0] := 84;
	Bounds[1] := 84;
	Bounds[2] := 72;
	Bounds[3] := 40;
	Bounds[4] := 40;
END_IF

button :=argButton;
fixer :=argFixer;
approx :=argApprox;
END_METHOD

END_FUNCTION_BLOCK

// ---- POUs/Stations/HRASI/InitAndTaskControl/RunInitClamperAndIndexer.TcPOU
FUNCTION_BLOCK RunInitClamperAndIndexer EXTENDS RunUnitGeneric
VAR_INPUT
	indexer : POINTER TO RunPnueIndexer;
	clampers : ARRAY[0..1] OF POINTER TO RunClamper;
	aoi : POINTER TO RunAoiInspectionV1;
	loader : POINTER TO runloading;
	
	okbin : POINTER TO RunBin;
	ngbin : POINTER TO RunBin;
	
	dimmer : POINTER TO RunUnitGeneric;
END_VAR
VAR_OUTPUT
END_VAR
VAR
	nCounter : INT;
END_VAR

SUPER^();

CASE outputState OF 
	eSpecialStates.INITIAL_BEGIN:
		bSerialTransition:=TRUE;
		FOR nCounter:=0 TO 1 BY 1 DO
			bSerialTransition := bSerialTransition AND clampers[nCounter]^.Initialize();
		END_FOR
		bSerialTransition := bSerialTransition AND aoi^.Initialize();
		bSerialTransition := bSerialTransition AND loader^.Initialize();
		bSerialTransition := bSerialTransition AND okbin<>0 AND_THEN okbin^.Initialize();
		bSerialTransition := bSerialTransition AND ngbin<>0 AND_THEN ngbin^.Initialize();
		bSerialTransition := bSerialTransition AND dimmer<>0 AND_THEN dimmer^.Initialize();
		
	eSpecialStates.INITIAL_STATE_1:
		bSerialTransition := indexer^.Initialize();
		IF bSerialTransition THEN
			NextState := eSpecialStates.INITIAL_END;
		END_IF
	//-----------------------
	//	Working
	//-----------------------
	eSpecialStates.GENERIC_GROUP_START:
		FOR nCounter:=0 TO 1 BY 1 DO
			clampers[nCounter]^.NextState := eSpecialStates.GENERIC_GROUP_START;
		END_FOR
		aoi^.NextState := eSpecialStates.GENERIC_GROUP_START;
		indexer^.NextState := eSpecialStates.GENERIC_GROUP_START;
		loader^.NextState := eSpecialStates.GENERIC_GROUP_START;
		
		ngbin^.NextState := eSpecialStates.GENERIC_GROUP_START;
		okbin^.NextState := eSpecialStates.GENERIC_GROUP_START;
		dimmer^.NextState := eSpecialStates.GENERIC_GROUP_START;
		
		bSerialTransition := TRUE; //into void state
END_CASE

END_FUNCTION_BLOCK

// ---- POUs/Stations/HRASI/RunPnueIndexer.TcPOU
FUNCTION_BLOCK RunPnueIndexer EXTENDS RunUnitIndexerMaster
VAR_INPUT
	sensorPairs : ARRAY[0..3] OF defSensorPair; //define stations sensor flag signatures
	fixtures : helperOutputSelection;
END_VAR
VAR_OUTPUT
END_VAR
VAR
	//devices
	lockCylinder : POINTER TO RunCylinder;
	pistonCylinder : POINTER TO RunCylinder;
	
	
	
	//----------------
	//	Initialization
	//----------------
	revolveCounter : INT;
	tickTime  AT%Q* : DWORD; 
	temp : bool;
END_VAR
VAR PERSISTENT
	revolveGoal : INT;
END_VAR

SUPER^(); //run indexer master

tickTime := TIME_TO_DWORD(workingTimerCache);

CASE outputState OF
	//---------------------------
	//	Initialization : revolve n times
	//---------------------------	
	eSpecialStates.INITIAL_BEGIN:
		revolveCounter:=0;
		bSerialTransition := TRUE;
	eSpecialStates.INITIAL_STATE_1:
		bSerialTransition := lockCylinder^.Execute(eCylinderCommands.COMMAND_B);
	eSpecialStates.INITIAL_STATE_2:
		bSerialTransition := pistonCylinder^.Execute(eCylinderCommands.COMMAND_B);
	eSpecialStates.INITIAL_STATE_3:
		bSerialTransition := lockCylinder^.Execute(eCylinderCommands.COMMAND_A);
	eSpecialStates.INITIAL_STATE_4:
		bSerialTransition := pistonCylinder^.Execute(eCylinderCommands.COMMAND_A);
		IF bSerialTransition THEN
			revolveCounter := revolveCounter+1;
			IF revolveCounter < revolveGoal THEN
				NextState := eSpecialStates.INITIAL_STATE_1; //repeat
			ELSE
				NextState := eSpecialStates.INITIAL_STATE_5; //to lock
			END_IF	
		END_IF
	eSpecialStates.INITIAL_STATE_5:
		bSerialTransition := lockCylinder^.Execute(eCylinderCommands.COMMAND_B);
		IF bSerialTransition THEN
			
			FOR nCounter :=0 TO SlotCount-1 BY 1 DO
				SlotBase[nCounter].Valid := FALSE; //reset
			END_FOR
			
			NextState := eSpecialStates.INITIAL_END; //terminated
		END_IF
	//------------------start running
	// S16#10 - : setup vacuum fixtures
	// S16#20 - : pnuematic indexer movement
	// 1. unlock
	// 2. shift out
	// 3. lock
	//------------------
	16#10:
		//activate fixture by slot valid status
		FOR nCounter := 0 TO SlotCount-1 BY 1 DO
			fixtures.Trigger(sensorPairs[nCounter],SlotBase[nCounter].Valid); 
		END_FOR
		NextState := 16#20;
	//----------
	16#20:
		bSerialTransition := pistonCylinder^.Execute(eCylinderCommands.COMMAND_B) ;
	16#21:
		bSerialTransition := lockCylinder^.Execute(eCylinderCommands.COMMAND_A);
	16#22:
		bSerialTransition := pistonCylinder^.Execute(eCylinderCommands.COMMAND_A);
	16#23:
		bSerialTransition := lockCylinder^.Execute(eCylinderCommands.COMMAND_B);
		IF bSerialTransition THEN
			
			
		
			fixtures.ReleaseAll(); //release all fixture
			NextState := 16#0F; //join master sequence
		END_IF
END_CASE

METHOD FB_init : BOOL
VAR_INPUT
	bInitRetains : BOOL; // if TRUE, the retain variables are initialized (warm start / cold start)
	bInCopyCode : BOOL;  // if TRUE, the instance afterwards gets moved into the copy code (online change)
	
	argParent : POINTER TO RunUnitGeneric;
	argSlotBase : POINTER TO RunMaterial;
	argSlotLast : POINTER TO RunMaterial;
	
	argUpstream : POINTER TO RunUnitTransporterBase;
	argAxis : POINTER TO RunAxis;
	
	argLockCylinder : POINTER TO RunCylinder;
	argPistonCylinder : POINTER TO RunCylinder;
END_VAR
//initialize 
Parent := argParent;
SlotBase := argSlotBase;
SlotLast := argSlotLast;

Axis := argAxis;
Upstream := argUpstream;

isProxyMode:=FALSE; //no proxy


//calculate how much slot related
SlotCount :=  TO_INT((SlotLast-SlotBase)/SIZEOF(RunMaterial) + 1);

lockCylinder := argLockCylinder;
pistonCylinder := argPistonCylinder;
END_METHOD

METHOD Initialize : BOOL
VAR_INPUT
END_VAR
VAR
	nCounter : int;
END_VAR
//once initializing method call , redirect current state to initalizing region
IF (TO_UINT(State) AND TO_UINT(eSpecialStates.INITIAL_REGION)) =0 THEN
	NextState := eSpecialStates.INITIAL_BEGIN; //not in intializing region , change
END_IF

Initialize := (State = eSpecialStates.INITIAL_END);

IF Initialize THEN
	//clear all remained signal
	FOR nCounter:=1 TO 32 BY 1 DO
		slaveWorkingSignal[nCounter] := FALSE;
	END_FOR
	//clear all internal status
	bEnStep := FALSE;
	bTrigStep := FALSE;
	bIsBypassed := FALSE;
	bWorkingOverride := FALSE;
	bMaterialOverride := FALSE;	
END_IF
END_METHOD

END_FUNCTION_BLOCK

// ---- POUs/Stations/HRASI/RunBin.TcPOU
FUNCTION_BLOCK RunBin EXTENDS RunUnitGeneric
VAR_INPUT
	sensor : POINTER TO RunSignal;
	ack AT%I* : BOOL;
	collectionCount AT%M*: UDINT;
END_VAR
VAR_OUTPUT
	ready AT%Q* : BOOL;
END_VAR
VAR	
	tickTime AT%Q*: DWORD ; //in ms
	
	totalCount AT%M* : UDINT; //wonld't be reset for each batch
END_VAR
VAR PERSISTENT
	collectionLimit AT%M* : UINT;
END_VAR

SUPER^();

//------------------
//the "READY" status
//------------------ 
ready := (collectionCount < collectionLimit) AND  (sensor <> 0 AND_THEN sensor^.debouncedOn) AND NOT ack;
IF NOT ready AND (collectionCount <> 0 AND (sensor <> 0 AND_THEN  sensor^.debouncedOff)) THEN
	collectionCount := 0; //count reset
END_IF
IF NOT ready AND NOT timeoutTimer.IN THEN
	timeoutTimer.IN := TRUE;
ELSIF NOT ready AND  timeoutTimer.Q  AND AlarmCode=0 THEN
	WarningCode := eErrorReasons.ERR_IDLE;
ELSIF ready THEN
	WarningCode := 0;
	timeoutTimer.IN := FALSE;
END_IF

CASE outputState OF
	eSpecialStates.INITIAL_BEGIN:
		collectionCount := 0;
		NextState := eSpecialStates.INITIAL_END;
	//-----------------
	//	START
	//-----------------
	eSpecialStates.GENERIC_GROUP_START:
		bSerialTransition := ack;
		IF bSerialTransition THEN
			
			//tick time calculation
			tickTime := TIME_TO_DWORD(workingTimer.ET);
			workingTimer.IN := FALSE;
		
			collectionCount := IncNoOverflow(input:= collectionCount);
			totalCount := IncNoOverflow(input:= totalCount);
			
		END_IF
	1: 
		bSerialTransition := NOT ack;
		IF bSerialTransition THEN
			NextState := eSpecialStates.GENERIC_GROUP_START;
		END_IF
END_CASE

END_FUNCTION_BLOCK

// ---- POUs/Stations/HRASI/InitAndTaskControl/RunInitScaraAndRack.TcPOU
FUNCTION_BLOCK RunInitScaraAndRack EXTENDS RunUnitGeneric
VAR_INPUT
	scara : POINTER TO RunScaraAgent;
	racks : ARRAY[0..1] OF POINTER TO RunCommonRack;
	bridges : ARRAY[0..3] OF POINTER TO RunBridge;
END_VAR
VAR_OUTPUT
END_VAR
VAR
	nCounter : INT;
END_VAR

SUPER^();



CASE outputState OF 
	eSpecialStates.INITIAL_BEGIN:
		bSerialTransition := scara^.Initialize();
	eSpecialStates.INITIAL_STATE_1:
		bSerialTransition := TRUE;
		FOR nCounter:=0 TO 1 BY 1 DO
			bSerialTransition := bSerialTransition AND racks[nCounter]^.Initialize();
		END_FOR
	eSpecialStates.INITIAL_STATE_2:
		bSerialTransition := TRUE;
		FOR nCounter:=0 TO 3 BY 1 DO
			IF bridges[nCounter]<>0 THEN
				bSerialTransition := bSerialTransition AND bridges[nCounter]^.Initialize();
			END_IF	
		END_FOR
		IF bSerialTransition THEN
			NextState := eSpecialStates.INITIAL_END; //ready for action
		END_IF
	//---------------------
	//	Then start working
	//---------------------
	eSpecialStates.GENERIC_GROUP_START:
		scara^.NextState := eSpecialStates.GENERIC_GROUP_START; //start working
		FOR nCounter:=0 TO 1 BY 1 DO
			racks[nCounter]^.NextState := eSpecialStates.GENERIC_GROUP_START;
		END_FOR
		FOR nCounter:=0 TO 3 BY 1 DO
			IF bridges[nCounter]<>0 THEN
				bridges[nCounter]^.NextState := eSpecialStates.GENERIC_GROUP_START;
			END_IF	
		END_FOR
		bSerialTransition := TRUE; // to void state
END_CASE

END_FUNCTION_BLOCK

// ---- POUs/Stations/HRASI/RunDimmerControl.TcPOU
FUNCTION_BLOCK RunDimmerControl EXTENDS RunUnitGeneric
VAR_INPUT
	mode : INT; //idle = 0, commissioning = 1(switch mode change is forbidden);
END_VAR
VAR_OUTPUT
END_VAR
VAR
	bCommandChanged : BOOL;	

	//Application layer
	//intesity-command,
	//intesity-ack
	command_intensity : ARRAY[0..7] OF BYTE;
	command_mode : ARRAY[0..7] OF BOOL;
	
	//mode-command,
	//mode-ack,
	status_intensity : ARRAY[0..7] OF BYTE;
	status_mode : ARRAY[0..7] OF BOOL;

	// I/O layer
	// (* I/O variables for a PC-COM port *)
    stIn_PcCom AT %I* : PcComInData; (* linked to the port in the TwinCAT System Manager *)
    stOut_PcCom AT %Q* : PcComOutData; (* linked to the port in the TwinCAT System Manager *)
    RxBufferPcCom  : ComBuffer; (* Receive data buffer; used with all receive function blocks *)
    TxBufferPcCom : ComBuffer; (* Transmit data buffer; used with all receive function blocks *)
	
	fbPcComCtrl			: SerialLineControl; // Gate to communicate with I/O layer
	bPcComCtrlError: BOOL;
	ePcComCtrlErrorID	: ComError_t;
	
	// Upper layer
	command : INT;
	
	dataSend : ARRAY[0..15] OF BYTE;
	
	dataPrefix : BYTE;
	dataSufix : byte;
	dataReceive : ARRAY[0..15] OF BYTE;
	
	
	fbSend : SendData;
	fbReceive : ReceiveData;
	
	timer : TON;
	
	nCounter : INT;
	queryCounter :BYTE;  // 0: ask mode, 1-channelNum : ask intensity
END_VAR
VAR CONSTANT
	BYTE_0_PRE : INT := 0;
	BYTE_1_REQ_ACK : INT := 1;
	BYTE_2_OPT : INT := 2;
	BYTE_3_POST : INT :=3;	

	DATA_PREFIX : BYTE := 16#FF;
	DATA_POSTFIX : BYTE := 16#FE;
	
	DATA_QUERY : BYTE := 16#12;
	
	DATA_REQ_MODE_HEAD : BYTE := 16#09;
	DATA_REQ_INTENSITY_HEAD : BYTE := 16#01;
	
	DATA_ACK_MODE : BYTE := 16#0;
	
END_VAR
VAR PERSISTENT
	channelNum : INT := 4;	
END_VAR



//initialize , query current status and intensity


//command , send when application variable changed

//routine-query
CASE outputState OF
	
	//----------------------------
	//	Working
	//----------------------------
	eSpecialStates.SLAVE_ENTER_PROCEDURE:
		//IDLE , check if command changed compared to status
		bCommandChanged := FALSE;
		
		IF mode=0 THEN
			//scan configuration 
			FOR nCounter :=0 TO channelNum DO
				IF NOT bSerialTransition THEN
					bSerialTransition := (command_mode[nCounter] <> status_mode[nCounter]);
					dataSend[BYTE_1_REQ_ACK] := DATA_REQ_MODE_HEAD;	
					dataSend[BYTE_2_OPT] :=  TO_BYTE(command_mode[nCounter]);
					queryCounter := 0;
				END_IF		
			END_FOR
		END_IF
		//scan if intensity changed
		FOR nCounter :=0 TO channelNum DO
			IF NOT bSerialTransition THEN
				bSerialTransition :=(command_intensity[nCounter] <> status_intensity[nCounter]);
				dataSend[BYTE_1_REQ_ACK] := DATA_REQ_INTENSITY_HEAD;	
				dataSend[BYTE_2_OPT] :=  command_intensity[nCounter];
				queryCounter := TO_BYTE(nCounter +1); // channel no.
			END_IF			
		END_FOR
		
		IF bCommandChanged THEN
			//------------------
			// Command Preparation
			//------------------
		END_IF
		
		// change dataSend to Query or Command
		IF bSerialTransition THEN
			timer.IN := TRUE;
		END_IF
				
	
		
		
	16#202:
		// Sender
		IF timer.Q THEN
			fbSend(pSendData := ADR(datasend),
				Length := SIZEOF(datasend),
				TXbuffer := TxBufferPcCom);
			timer.IN := FALSE; // reset
		END_IF
		IF timer.Q AND fbSend.Error = ComError_t.COMERROR_NOERROR AND NOT fbSend.Busy THEN
			bSerialTransition := TRUE;
		ELSIF timer.Q AND NOT fbSend.Busy AND fbSend.Error <> ComError_t.COMERROR_NOERROR THEN
			timer.IN := TRUE; // restart
		END_IF
	
	16#201:
		
		
		IF queryCounter < channelNum THEN
			// send
			bSerialTransition := TRUE;
		ELSE
			//------------------
			// Query Preparation
			//------------------
			dataSend[BYTE_1_REQ_ACK] := DATA_QUERY;		
			dataSend[BYTE_2_OPT] := queryCounter;
			NextState := 16#202;
		END_IF
		
END_CASE

//Receiver dispatcher
fbReceive(pPrefix := ADR(dataPrefix),
	LenPrefix:=to_byte(sizeof(dataPrefix)),
	pSuffix:=ADR(dataSufix),
	lensuffix:=to_byte(sizeof(dataSufix)),
	pReceiveData:=ADR(dataReceive),
	SizeReceiveData:=SIZEOF(dataReceive),	
RXbuffer:=RxBufferPcCom);

IF fbReceive.DataReceived THEN
	// process incoming message
	IF dataReceive[BYTE_1_REQ_ACK] = 0 THEN
		// MODE , update mode status
		FOR nCounter:=0 TO channelNum DO
			status_mode[nCounter] := (dataReceive[BYTE_2_OPT] AND SHL(16#01,nCounter)) <> 0;
		END_FOR
	ELSIF dataReceive[BYTE_1_REQ_ACK] <= channelNum THEN
		// Intensity , update intensity status , valid if within channel number
		status_intensity[dataReceive[BYTE_1_REQ_ACK]] := dataReceive[BYTE_2_OPT];
	END_IF
	
	//afterward , clean receiving buffer
	FOR nCounter:=0 TO SIZEOF(dataReceive)-1 DO
		dataReceive[nCounter]:=0;
	END_FOR
	
ELSE
	// Receiving	
END_IF


//----------------
// I/O Routine
//-----------------
fbPcComCtrl(
	Mode:= SERIALLINEMODE_PC_COM_PORT, 
	pComIn:= ADR(stIn_PcCom), 
	pComOut:= ADR(stOut_PcCom), 
	SizeComIn:= SIZEOF(stIn_PcCom), 
	Error=> , 
	ErrorID=> , 
	TxBuffer:= TxBufferPcCom, 
	RxBuffer:= RxBufferPcCom );
IF fbPcComCtrl.Error THEN
	bPcComCtrlError := TRUE;
	ePcComCtrlErrorID := fbPcComCtrl.ErrorID;
END_IF

END_FUNCTION_BLOCK

// ---- POUs/Stations/RunAoiHandshaking.TcPOU
FUNCTION_BLOCK RunAoiHandshaking EXTENDS RunUnitSlave
VAR_INPUT
	isLastShot : BOOL;
END_VAR
VAR
	registers : ARRAY[0..127] OF WORD; // memory poll to modbus server
	//pointers
	motionOnline : POINTER TO WORD := ADR(registers[indexMotionOnline]);
	motionTrigger: POINTER TO WORD := ADR(registers[indexMotionTrigger]);
	aoiOnline: POINTER TO WORD := ADR(registers[indexAoiOnline]);
	aoiAcknowledge: POINTER TO WORD := ADR(registers[indexAoiAcknowledge]);
	//-----------------------------------
	aoiData0 : POINTER TO MaterialBlock := ADR(registers[indexAoiData0]);
	//-----------------------------------
END_VAR
VAR CONSTANT
	indexMotionOnline : INT := 0;
	indexMotionTrigger : INT :=1;
	indexAoiOnline : INT := 4;
	indexAoiAcknowledge : INT :=5;
	indexAoiData0 : INT :=32;
END_VAR
VAR PERSISTENT	
	timeoutTimer : TON;
END_VAR

SUPER^();

//set motion offline once bypassed
IF bIsBypassed THEN
	motionOnline^ := 0;
ELSE
	motionOnline^ := 1;
END_IF

timeoutTimer(IN:= , PT:= , Q=> , ET=> );
IF NOT timeoutTimer.IN THEN
	timeoutTimer.IN := TRUE;
END_IF

CASE outputState OF
	eSpecialStates.SLAVE_ENTER_PROCEDURE:
		aoiData0^.data[0] := 16#FF;//set 0xff to AOI_DATA_0 as marker
		IF NOT bIsBypassed THEN
			//go ahead
			motionTrigger^ := 1;
			//aoiAcknowledge^ := 0; //auto reset
			bSerialTransition := TRUE;
		ELSE
			//bypassed
			NextState := 16#300;
		END_IF
	16#201:
		//check AOI acknowledged
		IF aoiAcknowledge^ = 1 THEN
			motionTrigger^ := 0;
			bSerialTransition := TRUE;
			
			//inform motion to do next position ahead the handshaking procedure
			workingSignal^ := FALSE;
			
		ELSIF timeoutTimer.Q THEN
			//timeout warning
		END_IF
	16#202:
		//wait until AOI_DATA write-in once last shot
		transitionByte.0 := (aoiAcknowledge^=0) AND (NOT isLastShot OR (isLastShot AND aoiData0^.data[0] <> 16#FF));
		IF transitionByte.0 THEN
			NextState := 16#300;
		ELSIF timeoutTimer.Q THEN
			//timeout warning
		END_IF
	//-----------------------------------
	16#300:
		//move data to Slot
		SlotBase^.Data := aoiData0^;
		
		//trigger Database communiction
		IF isLastShot THEN
			SlotBase^.Act := TRUE;
		END_IF
		
		NextState := 0;
END_CASE

IF bSerialTransition OR NextState<>outputState THEN
	timeoutTimer.IN := FALSE; //reset
END_IF

//once AOI_Offline detected , to bypass
IF NOT aoiOnline^=1 AND NOT bIsBypassed THEN
	bIsBypassed := TRUE;
	motionTrigger^ := 0;	//reset motion trigger
	aoiData0^.data[0] := 0; //OK/NG data reset
	NextState := 16#300;
END_IF

METHOD Initialize : BOOL
VAR_INPUT
END_VAR
CASE outputState OF
	eSpecialStates.INITIAL_BEGIN:		
			NextState := eSpecialStates.INITIAL_END;
END_CASE

Initialize := SUPER^.Initialize();
END_METHOD

END_FUNCTION_BLOCK

// ---- POUs/Stations/RunAxisAoiView.TcPOU
FUNCTION_BLOCK RunAxisAoiView EXTENDS RunAxisInspection
VAR
	
END_VAR

SUPER^();

CASE outputState OF
	eSpecialStates.SLAVE_ENTER_PROCEDURE:
		IF bMaterialOverride THEN
			bSerialTransition := TRUE;
		ELSE
			NextState := eSpecialStates.SLAVE_WORK_DONE;
		END_IF
	16#201:
		//align
		IF sideAligner^.Execute(argCommand:= eCylinderCommands.COMMAND_B) THEN
			NextState := eSpecialStates.SLAVE_AXIS_INSPECTION_ENTER;
		END_IF
	//----------------------------------
	eSpecialStates.SLAVE_AXIS_INSPECTION_EXIT:
		//release
		IF NOT transitionByte.0 AND_THEN axis1^.ExecuteParameterIndex(indexStandByAxis1) THEN
			transitionByte.0 := TRUE;
		END_IF
		IF NOT transitionByte.1 AND_THEN (axis2 = 0 OR axis2<>0 AND_THEN axis2^.ExecuteParameterIndex(indexStandByAxis2)) THEN
			transitionByte.1 := TRUE; //axis 2 is not existed
		END_IF	
		IF NOT transitionByte.2 AND_THEN sideAligner^.Execute(eCylinderCommands.COMMAND_A) THEN
			transitionByte.2 := TRUE;
		END_IF
		IF transitionByte = 7 THEN
			NextState := eSpecialStates.SLAVE_WORK_DONE;
		END_IF
END_CASE

METHOD Initialize : BOOL
VAR_INPUT
END_VAR
//default initialization sequence
CASE outputState OF 
	eSpecialStates.INITIAL_BEGIN:
		NextState := eSpecialStates.INITIAL_STATE_7;
END_CASE

Initialize := SUPER^.Initialize();
END_METHOD

END_FUNCTION_BLOCK

// ---- POUs/Stations/RunAxisInspection.TcPOU
FUNCTION_BLOCK RunAxisInspection EXTENDS RunUnitSlave
VAR
	axis1 : POINTER TO RunAxis;
	axis2 : POINTER TO RunAxis;
	sideAligner : POINTER TO RunCylinder := 0;
	
	nCounter : INT := 0;
END_VAR
VAR_OUTPUT
	isLastShot : BOOL;
END_VAR
VAR PERSISTENT
	//Axis1
	indexStandByAxis1 : INT := 1;
	indexPosition1Axis1 : INT := 2;
	//Axis2
	indexStandByAxis2 : INT := 1;
	indexPosition1Axis2 : INT := 2;
	//
	nGoal : INT := 4;
END_VAR

//n-Axis aoi , once position completed , trigger and wait
SUPER^();

CASE outputState OF
	eSpecialStates.SLAVE_AXIS_INSPECTION_ENTER:
		IF NOT transitionByte.0 THEN
			transitionByte.0 := axis1^.ExecuteParameterIndex(nCounter + indexPosition1Axis1);
		END_IF
		IF NOT transitionByte.1 AND_THEN (axis2 = 0 OR (axis2<>0 AND_THEN axis2^.ExecuteParameterIndex(nCounter + indexPosition1Axis2))) THEN
			transitionByte.1 := TRUE; // axis2 is not existed or // axis2 is existed
		END_IF
		IF transitionByte = 3 THEN
			//once inspection done
			NextState := eSpecialStates.SLAVE_AXIS_INSPECTION_ITERATION; //both axis done motion
			slaveWorkingSignal[1] := slaveLinkageStatus[1]; //trigger slave
		END_IF
	eSpecialStates.SLAVE_AXIS_INSPECTION_ITERATION:
		IF NOT slaveWorkingSignal[1] THEN
			//once inspection reach 
			IF nCounter < nGoal THEN			
				nCounter := nCounter + 1;
				NextState := eSpecialStates.SLAVE_AXIS_INSPECTION_ENTER;
			ELSE
				//greater and equal goal
				nCounter := 0; //reset
				NextState := eSpecialStates.SLAVE_AXIS_INSPECTION_EXIT;
			END_IF
		ELSE
			//wait inspecition
		END_IF
END_CASE

//reflect
isLastShot := (nCounter = nGoal);

METHOD FB_init : BOOL
VAR_INPUT
	bInitRetains : BOOL; // if TRUE, the retain variables are initialized (warm start / cold start)
	bInCopyCode : BOOL;  // if TRUE, the instance afterwards gets moved into the copy code (online change)
	
	argParent : POINTER TO RunUnitGeneric;
	argSlotBase : POINTER TO RunMaterial;
	argSlotLast : POINTER TO RunMaterial;
	
	argWorkingSignal : POINTER TO BOOL;
	
	argAxis1 : POINTER TO RunAxis;
	argAxis2 : POINTER TO RunAxis;
	
	argSideAligner : POINTER TO RunCylinder;
END_VAR
//initialize 
Parent := argParent;
SlotBase := argSlotBase;
SlotLast := argSlotLast;
//
IF bInitRetains THEN
	NextState := eSpecialStates.INITIAL_BEGIN;
END_IF

workingSignal := argWorkingSignal; //link

axis1 := argAxis1;
axis2 := argAxis2;
sideAligner := argSideAligner;
END_METHOD

METHOD Initialize : BOOL
VAR_INPUT
END_VAR

//default initialization sequence
CASE outputState OF 
	eSpecialStates.INITIAL_STATE_7:
		IF NOT transitionByte.0 AND_THEN axis1^.ExecuteParameterIndex(indexStandByAxis1) THEN
			transitionByte.0 := TRUE;
		END_IF
		IF NOT transitionByte.1 AND_THEN (axis2 = 0 OR axis2<>0 AND_THEN axis2^.ExecuteParameterIndex(indexStandByAxis2)) THEN
			transitionByte.1 := TRUE; //axis 2 is not existed
		END_IF
		IF NOT transitionByte.2 AND_THEN (sideAligner=0 OR (sideAligner<>0 AND_THEN sideAligner^.Execute(eCylinderCommands.COMMAND_A))) THEN
			transitionByte.2 := TRUE; //aligner backoff
		END_IF
		IF transitionByte = 7 THEN
			nCounter:=0;//reset
			NextState := eSpecialStates.INITIAL_END;
		END_IF
END_CASE

Initialize:= SUPER^.Initialize();
END_METHOD

END_FUNCTION_BLOCK

// ---- POUs/Stations/RunBottomView.TcPOU
FUNCTION_BLOCK RunBottomView EXTENDS RunAxisInspection
VAR_INPUT
END_VAR
VAR_OUTPUT
END_VAR
VAR
	connectorHolder : POINTER TO RunCylinder; //also the cable holder
	transporter : POINTER TO RunCylinder;
	openClamp : POINTER TO RunCylinder;
END_VAR
VAR PERSISTENT
	indexCommandReadyPick : int;
	indexCommandPick : INT;
END_VAR

SUPER^();

CASE outputState OF
	eSpecialStates.SLAVE_ENTER_PROCEDURE:
		IF bMaterialOverride THEN
			bSerialTransition := TRUE;
		ELSE
			NextState := eSpecialStates.SLAVE_WORK_DONE;
		END_IF
	16#201:
		bSerialTransition := axis1^.ExecuteParameterIndex(indexCommand:= indexCommandPick); //down
	16#202:
		bSerialTransition:=connectorHolder^.Execute(argCommand:= eCylinderCommands.COMMAND_B); //hold
	16#203:
		bSerialTransition:=openClamp^.Execute(argCommand:= eCylinderCommands.COMMAND_B); //release
	16#204:
		bSerialTransition:=axis1^.ExecuteParameterIndex(indexCommand:= indexStandByAxis1); //up ( standby position should not interfere with cam
	16#205:
		//go to inspection 1 simulatanously
		IF NOT transitionByte.0 AND_THEN transporter^.Execute(argCommand:= eCylinderCommands.COMMAND_B) THEN
			transitionByte.0 := TRUE;
		END_IF
		IF NOT transitionByte.1 AND_THEN axis2^.ExecuteParameterIndex(indexCommand:= indexStandByAxis2) THEN
			//axis2 : CCD moving carriage
			transitionByte.1 := TRUE;
		END_IF
		IF transitionByte=3 THEN
			NextState := eSpecialStates.SLAVE_AXIS_INSPECTION_ENTER;
		END_IF
	//----------------------Return
	eSpecialStates.SLAVE_AXIS_INSPECTION_EXIT:
		//up ( standby position should not interfere with cam
		IF axis1^.ExecuteParameterIndex(indexCommand:= indexStandByAxis1) THEN
			NextState := 16#500;
		END_IF
	//----------------------
	16#500:
		//return simulatanously
		IF NOT transitionByte.0 AND_THEN transporter^.Execute(argCommand:= eCylinderCommands.COMMAND_A) THEN
			transitionByte.0 := TRUE;
		END_IF
		IF NOT transitionByte.1 AND_THEN axis2^.ExecuteParameterIndex(indexCommand:= indexStandByAxis2) THEN
			transitionByte.1 := TRUE;
		END_IF
		IF transitionByte=3 THEN
			NextState := 16#501;
		END_IF
	16#501:
		bSerialTransition:=axis1^.ExecuteParameterIndex(indexCommand:= indexCommandPick);//down
	16#502:
		bSerialTransition:=connectorHolder^.Execute(argCommand:= eCylinderCommands.COMMAND_A); //release
	16#503:
		bSerialTransition:=openClamp^.Execute(argCommand:= eCylinderCommands.COMMAND_A); //hold
	16#504:
		IF axis1^.ExecuteParameterIndex(indexCommand:= indexCommandReadyPick) THEN
			NextState := eSpecialStates.SLAVE_WORK_DONE;
		END_IF
END_CASE

METHOD FB_init : BOOL
VAR_INPUT
	bInitRetains : BOOL; // if TRUE, the retain variables are initialized (warm start / cold start)
	bInCopyCode : BOOL;  // if TRUE, the instance afterwards gets moved into the copy code (online change)
	
	argParent : POINTER TO RunUnitGeneric;
	argSlotBase : POINTER TO RunMaterial;
	argSlotLast : POINTER TO RunMaterial;
	
	argWorkingSignal : POINTER TO BOOL;
	
	argAxis1 : POINTER TO RunAxis;
	argAxis2 : POINTER TO RunAxis;
	
	argSideAligner : POINTER TO RunCylinder;
	
	argConnectorHolder : POINTER TO RunCylinder;
	argTransporter : POINTER TO RunCylinder;
	argOpenClamp : POINTER TO RunCylinder;
END_VAR
//initialize 
Parent := argParent;
SlotBase := argSlotBase;
SlotLast := argSlotLast;
//
IF bInitRetains THEN
	NextState := eSpecialStates.INITIAL_BEGIN;
END_IF

workingSignal := argWorkingSignal; //link

axis1 := argAxis1;
axis2 := argAxis2;
sideAligner := 0;

connectorHolder := argConnectorHolder;
transporter := argTransporter;
openClamp := argOpenClamp;
END_METHOD

METHOD Initialize : BOOL
VAR_INPUT
END_VAR

CASE outputState OF
	eSpecialStates.INITIAL_BEGIN:
		// release all cylinder
		IF NOT transitionByte.0 AND_THEN connectorHolder^.Execute(argCommand:= eCylinderCommands.COMMAND_A) THEN
			transitionByte.0 := TRUE;
		END_IF
		IF NOT transitionByte.1 AND_THEN transporter^.Execute(argCommand:= eCylinderCommands.COMMAND_A) THEN
			transitionByte.1 := TRUE;
		END_IF
		IF NOT transitionByte.2 AND_THEN openClamp^.Execute(argCommand:= eCylinderCommands.COMMAND_A) THEN
			transitionByte.2 := TRUE;
		END_IF
		IF transitionByte=7 THEN
			NextState := eSpecialStates.INITIAL_STATE_1; // to return axis
		END_IF
	eSpecialStates.INITIAL_STATE_1:
		IF NOT transitionByte.0 AND_THEN axis1^.ExecuteParameterIndex(indexCommand:= indexCommandReadyPick) THEN
			transitionByte.0 := TRUE;
		END_IF
		IF NOT transitionByte.1 AND_THEN axis2^.ExecuteParameterIndex(indexCommand:= indexStandByAxis2)THEN
			transitionByte.1 := TRUE;
		END_IF
		IF transitionByte = 3 THEN
			NextState := eSpecialStates.INITIAL_END;
		END_IF
END_CASE

//once initializing method call , redirect current state to initalizing region
IF (TO_UINT(State) AND TO_UINT(eSpecialStates.INITIAL_REGION)) =0 THEN
	NextState := eSpecialStates.INITIAL_BEGIN; //not in intializing region , change
END_IF

Initialize := (State = eSpecialStates.INITIAL_END);

IF Initialize THEN
	//clear all remained signal
	FOR nCounter:=1 TO 32 BY 1 DO
		slaveWorkingSignal[nCounter] := FALSE;
	END_FOR
	//clear all internal status
	bEnStep := FALSE;
	bTrigStep := FALSE;
	bIsBypassed := FALSE;
	bWorkingOverride := FALSE;
	bMaterialOverride := FALSE;	
END_IF
END_METHOD

END_FUNCTION_BLOCK

// ---- POUs/Stations/RunETest.TcPOU
FUNCTION_BLOCK RunETest EXTENDS RunAxisInspection
VAR
	
	//Cylinders
	connectorHolder : POINTER TO RunCylinder;
	cableHolder : POINTER TO RunCylinder;
	plugin : POINTER TO RunCylinder;
	//Sensors
	tongueExistedA : POINTER TO RunSignal;
	tongueExistedB : POINTER TO RunSignal;
	tongueGlueA : POINTER TO RunSignal;
	tongueGlueB : POINTER TO RunSignal;
	//from tester
	ioBundle : POINTER TO ioBundleET;
	//
	isOK : BOOL;
	isRedo : BOOL;
	etSeriesNgCounter : UINT;
	etRedoCounter : UINT;
	//
	block : MaterialBlock;
END_VAR
VAR PERSISTENT
	indexCommandPick : INT := 1;
	indexReleaseConnectorHolder : INT := 1;
	
	etUsageCounter : UINT;
	etUsageThreshold : UINT;
	
	etNgAlarmSwitch : BOOL;
	etSeriesNgThreshold : UINT;
	etRedoGoal : UINT;
END_VAR

SUPER^();

IF etUsageCounter>=etUsageThreshold THEN
	//!Clear by manual operation
	AlarmCode := eErrorCodes.AC_ET_USAGE_MEET; 
END_IF

CASE outputState OF
	eSpecialStates.SLAVE_ENTER_PROCEDURE:
		IF bMaterialOverride THEN
			bSerialTransition := TRUE;
		ELSE
			NextState := eSpecialStates.SLAVE_WORK_DONE;
		END_IF
	16#201:
		bSerialTransition := connectorHolder^.Execute(eCylinderCommands.COMMAND_B);
	16#202:
		bSerialTransition := plugin^.Execute(eCylinderCommands.COMMAND_B);
		IF bSerialTransition THEN
			//usage count-up
			etUsageCounter := etUsageCounter+1;
		END_IF
	16#203:
		bSerialTransition := axis1^.ExecuteParameterIndex(indexCommandPick); //down to pick
	16#204:
		bSerialTransition := cableHolder^.Execute(eCylinderCommands.COMMAND_B) ;//hold 
	16#205:
		IF TRUE THEN
			//going to swing
			NextState := eSpecialStates.SLAVE_AXIS_INSPECTION_ENTER;
		END_IF
	//-----------------
	eSpecialStates.SLAVE_AXIS_INSPECTION_EXIT:
		//TODO , read status and report
		isOK := tongueExistedA^.debouncedOn AND tongueExistedB^.debouncedOn AND  tongueGlueA^.debouncedOff AND tongueGlueB^.debouncedOff AND ioBundle^.o3;
		
		isRedo := FALSE;//reset
		IF isOK THEN
			//ok
			etSeriesNgCounter := 0;
		ELSE
			//ng
			etSeriesNgCounter := etSeriesNgCounter+1;
			IF 	(etSeriesNgCounter >= etSeriesNgThreshold) AND etNgAlarmSwitch AND (etRedoCounter >=etRedoGoal) THEN
				//raise alarm
				AlarmCode := eErrorCodes.AC_ET_SERIES_NG;
				etSeriesNgCounter := 0;
			ELSIF etRedoCounter < etRedoGoal THEN
				//not reach , redo
				isRedo := TRUE;
			END_IF
		END_IF		
		//report
		block.data[0] := TO_WORD(ioBundle^.o3); //et
		block.data[1] := TO_WORD(tongueExistedA^.debouncedOn);
		block.data[2] := TO_WORD(tongueExistedB^.debouncedOn);
		block.data[3] := TO_WORD(tongueGlueA^.debouncedOff);
		block.data[4] := TO_WORD(tongueGlueB^.debouncedOff);
		SlotBase^.Data := block;
		SlotBase^.Act := TRUE;
		
		bSerialTransition := TRUE;
	16#401:
		bSerialTransition := axis1^.ExecuteParameterIndex(indexCommandPick); //back to to pick
	16#402:
		bSerialTransition := cableHolder^.Execute(eCylinderCommands.COMMAND_A);
	16#403:
		bSerialTransition := plugin^.Execute(eCylinderCommands.COMMAND_A);
	16#404:
		bSerialTransition := connectorHolder^.Execute(eCylinderCommands.COMMAND_A);
	16#405:
		//all axis backto standby
		IF NOT transitionByte.0 AND_THEN axis1^.ExecuteParameterIndex(indexStandByAxis1) THEN
			transitionByte.0 := TRUE;
		END_IF
		IF NOT transitionByte.1 AND_THEN axis2^.ExecuteParameterIndex(indexStandByAxis2) THEN
			transitionByte.1 := TRUE;
		END_IF
		IF transitionByte=3 THEN
			IF isRedo THEN
				etRedoCounter := etRedoCounter+1;
				NextState := eSpecialStates.SLAVE_ENTER_PROCEDURE;
			ELSE
				etRedoCounter :=0; //reset
				NextState := eSpecialStates.SLAVE_WORK_DONE;
			END_IF
		END_IF
END_CASE
//release to swing // release connector holder when horizon moving
IF (slaveWorkingSignal[1] AND ((nCounter=indexReleaseConnectorHolder AND_THEN connectorHolder^.Execute(eCylinderCommands.COMMAND_A)) OR nCounter<>indexReleaseConnectorHolder)) THEN
	slaveWorkingSignal[1] := FALSE;
END_IF

METHOD FB_init : BOOL
VAR_INPUT
	bInitRetains : BOOL; // if TRUE, the retain variables are initialized (warm start / cold start)
	bInCopyCode : BOOL;  // if TRUE, the instance afterwards gets moved into the copy code (online change)
	
	argParent : POINTER TO RunUnitGeneric;
	argSlotBase : POINTER TO RunMaterial;
	argSlotLast : POINTER TO RunMaterial;
	
	argWorkingSignal : POINTER TO BOOL;
	
	argAxis1 : POINTER TO RunAxis;
	argAxis2 : POINTER TO RunAxis;
	
	argSideAligner : pointer to RunCylinder;
	
	argConnectorHolder : POINTER TO RunCylinder;
	argCableHolder : POINTER TO RunCylinder;
	argPlugin : POINTER TO RunCylinder;
	//Sensors
	argTongueExistedA : POINTER TO RunSignal;
	argTongueExistedB : POINTER TO RunSignal;
	argTongueGlueA : POINTER TO RunSignal;
	argTongueGlueB : POINTER TO RunSignal;
	
	argIoBundle : pointer to ioBundleET;
END_VAR
//initialize 
Parent := argParent;
SlotBase := argSlotBase;
SlotLast := argSlotLast;
//
IF bInitRetains THEN
	NextState := eSpecialStates.INITIAL_BEGIN;
END_IF

workingSignal := argWorkingSignal; //link

axis1 := argAxis1;
axis2 := argAxis2;

//
connectorHolder := argConnectorHolder;
cableHolder :=argCableHolder;
plugin :=argPlugin;
	//Sensors
tongueExistedA :=argTongueExistedA;
tongueExistedB :=argTongueExistedB;
tongueGlueA :=argTongueGlueA;
tongueGlueB :=argTongueGlueB;
ioBundle := argIoBundle;
END_METHOD

METHOD Initialize : BOOL
VAR_INPUT
END_VAR

CASE outputState OF
	eSpecialStates.INITIAL_BEGIN:
		// release all cylinder
		IF NOT transitionByte.0 AND_THEN plugin^.Execute(argCommand:= eCylinderCommands.COMMAND_A) THEN
			transitionByte.0 := TRUE;
		END_IF
		IF NOT transitionByte.1 AND_THEN connectorHolder^.Execute(argCommand:= eCylinderCommands.COMMAND_A) THEN
			transitionByte.1 := TRUE;
		END_IF
		IF NOT transitionByte.2 AND_THEN cableHolder^.Execute(argCommand:= eCylinderCommands.COMMAND_A) THEN
			transitionByte.2 := TRUE;
		END_IF
		IF transitionByte=7 THEN
			NextState := eSpecialStates.INITIAL_STATE_7; // to return axis
		END_IF
END_CASE


Initialize:= SUPER^.Initialize(); //do axis return
END_METHOD

END_FUNCTION_BLOCK

// ---- POUs/Stations/RunInputV1.TcPOU
FUNCTION_BLOCK RunInputV1 EXTENDS RunUnitSlave
VAR_INPUT
	handy : BOOL; //link to handy(on)
	lightScreen : BOOL; //link to light screen
		
	materialRemains : UINT; //link to the counter of all controllers
	
	materialValidSensor : BOOL; //link to approximity
END_VAR
VAR_OUTPUT
	inputCounter : UINT;
END_VAR
VAR
	clamper : POINTER TO RunCylinder;
	
	controller : POINTER TO RunUnitController; //link to parent
	toggleClear : BOOL; // link to HMI clear request
END_VAR

SUPER^();

//status backup
IF NOT toggleClear AND (controller<>0 AND_THEN controller^.interfaceControl^.materialClear) THEN
	toggleClear := TRUE;
END_IF

